	IF ( MsgRecBuffer[counter].MsgType = DATAREC AND   FIND(MsgRecBuffer[counter].Msg,  'NMEAS;MAC' ) = 4 ) AND ( FIND(MsgRecBuffer[counter].Msg,  'IDN' ) = 30) THEN
		StrSaveMacAdd:=MID(MsgRecBuffer[counter].Msg, 8 , 21);
		StrLoc:=33;
		Str := MID(MsgRecBuffer[counter].Msg, 1 , StrLoc);
		WHILE (SysStrCmp(Str,';')<>0 AND StrLoc<=255) DO (*Cerco il numero IDN e lo memorizzo in StrSaveID dopo il while*)
			StrLoc:=StrLoc+1;
			Str := MID(MsgRecBuffer[counter].Msg, 1 , StrLoc);
		END_WHILE
		StrSaveID:=MID(MsgRecBuffer[counter].Msg, StrLoc-33 , 33);
		index:=1;
		WHILE (index<=MAX_LUXNUM) AND (SysStrCmp(TabListLux[index].StMacAdd,  StrSaveMacAdd) <> 0)   DO (*diego setting *)
			index:= index +1;
		END_WHILE
		IF index<=MAX_LUXNUM AND STRING_TO_WORD(StrSaveID) >0 AND TabListLux[index].LuxID_Geolumen<>STRING_TO_WORD(StrSaveID)  THEN
			TabListLux[index].xCoupled := TRUE; (*Indico che ho accoppiato l'ID con il mac address*)
			TabListLux[index].LuxID_Geolumen:=STRING_TO_WORD(StrSaveID); (*Salvo l'ID accoppiato al mac address - info che sarà poi da spedire al server*)
			LuxElement[index].ID := TabListLux[index].LuxNumber; (*  copio id del lux nella tabella delle variabili dei lux *)
			IF LuxElement[index].CTRL_MODE = 2 THEN
				(* init astro *)
				ASTR[index](ID:= LuxElement[index].ID, localTime:=Sys.Time_CT_DT);
				ASTR_CONFIG[index].ID:=ASTR[index].ID;
			END_IF
			LuxGeolumenNodes[index].ID_Geolumen:=TabListLux[index].LuxID_Geolumen;
			LuxGeolumenNodes[index].ID_Lux:=TabListLux[index].LuxNumber;
			LuxGeolumenNodes[index].MAX_RETRY_NO_FEEDBACK:=MAX_RETRY_NO_FEEDBACK_GEOLUMEN_NODES;
			LuxGeolumenNodes[index].MAX_RETRY_STATUS_NOT_ALIGNED:=MAX_RETRY_STATUS_NOT_ALIGNED_GEOLUMEN_NODES;

			(*aggiorno stato*)
			parseNodeStatus(statusNodeMessage:=MsgRecBufferPtr^[counter].Msg);
			IF idNode>=1 AND idNode<=MAX_LUXNUM THEN
				tmpIndex:=getGeolumenNodeByGeolumenId (idNode);
				IF(tmpIndex>0 AND tmpIndex<=MAX_LUXNUM) THEN
					LuxGeolumenNodes[tmpIndex](feedbackState:=state); LuxGeolumenNodes[tmpIndex].updateFeedbackState();
				END_IF
			END_IF
		END_IF
	END_IF

	IF ( MsgRecBuffer[counter].MsgType = MED AND   FIND(MsgRecBuffer[counter].Msg,  'NMEASMED;MAC' ) = 4 ) AND ( FIND(MsgRecBuffer[counter].Msg,  'IDN' ) = 33) THEN
		StrSaveMacAdd:=MID(MsgRecBuffer[counter].Msg, 8 , 24);
		StrLoc:=36;
		Str := MID(MsgRecBuffer[counter].Msg, 1 , StrLoc);
		WHILE (SysStrCmp(Str,';')<>0 AND StrLoc<=255) DO (*Cerco il numero IDN e lo memorizzo in StrSaveID dopo il while*)
			StrLoc:=StrLoc+1;
			Str := MID(MsgRecBuffer[counter].Msg, 1 , StrLoc);
		END_WHILE
		StrSaveID:=MID(MsgRecBuffer[counter].Msg, StrLoc-36 , 36);
		index:=1;
		WHILE (index<=MAX_LUXNUM) AND (SysStrCmp(TabListLux[index].StMacAdd,  StrSaveMacAdd) <> 0)   DO (*diego setting *)
			index:= index +1;
		END_WHILE
		IF index<=MAX_LUXNUM AND STRING_TO_WORD(StrSaveID) >0 AND TabListLux[index].LuxID_Geolumen<>STRING_TO_WORD(StrSaveID)  THEN
			TabListLux[index].xCoupled := TRUE; (*Indico che ho accoppiato l'ID con il mac address*)
			TabListLux[index].LuxID_Geolumen:=STRING_TO_WORD(StrSaveID); (*Salvo l'ID accoppiato al mac address - info che sarà poi da spedire al server*)
			LuxElement[index].ID := TabListLux[index].LuxNumber; (*  copio id del lux nella tabella delle variabili dei lux *)
			IF LuxElement[index].CTRL_MODE = 2 THEN
				(* init astro *)
				ASTR[index](ID:= LuxElement[index].ID, localTime:=Sys.Time_CT_DT);
				ASTR_CONFIG[index].ID:=ASTR[index].ID;
			END_IF
			LuxGeolumenNodes[index].MAX_RETRY_NO_FEEDBACK:=MAX_RETRY_NO_FEEDBACK_GEOLUMEN_NODES;
			LuxGeolumenNodes[index].MAX_RETRY_STATUS_NOT_ALIGNED:=MAX_RETRY_STATUS_NOT_ALIGNED_GEOLUMEN_NODES;
			LuxGeolumenNodes[index].ID_Geolumen:=TabListLux[index].LuxID_Geolumen;
			LuxGeolumenNodes[index].ID_Lux:=TabListLux[index].LuxNumber;
		END_IF
	END_IF
END_ACTION
ACTION SendAuth:
(*...per compabilità indicizzazione Renato...*)
i:=ArrayPos-1;
IF(i<0) THEN i:=0; END_IF

(*TimerCmdAdd(IN:=NOT TimerCmdAdd.Q,PT:=T#5m);
IF TimerCmdAdd.Q THEN
	FOR x:= 1 TO MAX_LUXNUM DO
		TabListLuxSendAuth[x]:=0;
	END_FOR
END_IF*)


(*IF MsgRecBuffer[i].MsgType = REQAUTH0  THEN
	MacStr:=MID(MsgRecBuffer[i].Msg, 8, 23); (*Isolo la sottostringa del Mac address - es. 0046CD12*)

		FOR x:= 1 TO MAX_LUXNUM DO
			IF SysStrCmp(MacStr, TabListLux[x].StMacAdd) = 0 AND TabListLux[x].LuxID_Geolumen=0 AND TabListLuxSendAuth[x]<1 THEN
				TabListLuxSendAuth[x]:=TabListLuxSendAuth[x]+1;
				 (*spedisci autorizzazione   CMD_ADD_NODE:21:36096:70:50744$0D$0A  *)
				StrToSend:=CONCAT('LST_ADD_NODE:21,36096,', WORD_TO_STRING(TabListLux[x].MacAddH) );
				StrToSend:=CONCAT(StrToSend, ',');
				StrToSend:=CONCAT(StrToSend,  WORD_TO_STRING(TabListLux[x].MacAddL) );
				StrToSend:=CONCAT(StrToSend,  '$R' );
				(*SendData(pTxData:=ADR(StrToSend));*)
				SendDataQueue(pTxData:=ADR(StrToSend));
				SendDataQueue.addMessage();
				MsgRecBuffer[i].MsgType:=COMPLETED;
				x:=  MAX_LUXNUM+1;
			END_IF
		END_FOR

END_IF*)
END_ACTION
ACTION sendGlobalOff:
SendString := setGlobalOFF;
SendDataQueue(pTxData:=ADR(SendString));
SendDataQueue.addMessage();
END_ACTION
ACTION sendGlobalON:
SendString := setGlobalON;
SendDataQueue(pTxData:=ADR(SendString));
SendDataQueue.addMessage();
END_ACTION
ACTION updateNetworkTime:
(* creazione ed invio comando per settare orario della rete *)

StrMin:=BYTE_TO_STRING(Sys.Time_Min);
IF  Sys.Time_Min<=9 THEN
	StrMin := CONCAT('0',StrMin);
END_IF
StrMin:=MID(STR:=StrMin, LEN:=2, POS:= 1);
StrHour:=BYTE_TO_STRING(Sys.Time_Hour);
IF Sys.Time_Hour<=9 THEN
	StrHour := CONCAT('0',StrHour);
END_IF
StrHour:=MID(STR:=StrHour, LEN:=2, POS:= 1);

SendString := 'NWK_TIME_SET=$R';
SendString :=INSERT (SendString,StrHour,13);
SendString :=INSERT (SendString,':',15);
SendString :=INSERT (SendString,StrMin,16);

SendDataQueue(pTxData:=ADR(SendString));
SendDataQueue.addMessage();
END_ACTION

(* POU GeoLumenWrapping/SendDataQueue, ST *)
FUNCTION_BLOCK SendDataQueue
VAR CONSTANT
	QUEUE_SIZE:DWORD:=5000;
END_VAR
VAR_INPUT
	pTxData: POINTER TO STRING;
END_VAR
VAR_OUTPUT
	StrToSend: STRING;
	toBeSent : WORD:=0;
END_VAR
VAR
	writeIndex:DWORD:=0;
	readIndex:DWORD:=0;
	pRecStr 	: POINTER TO STRING(255);
	queue: ARRAY[1..QUEUE_SIZE] OF STRING(255);

END_VAR
;
END_FUNCTION_BLOCK
ACTION addMessage:
writeIndex:=((writeIndex+1) MOD (QUEUE_SIZE+1))+(writeIndex+1)/(QUEUE_SIZE+1);

queue[writeIndex]:=pTxData^;

IF(toBeSent<QUEUE_SIZE) THEN
	toBeSent:=toBeSent+1;
ELSE

	toBeSent:=1;

END_IF
END_ACTION
ACTION getMessage:
IF(toBeSent >0) THEN

	readIndex:=((readIndex+1) MOD (QUEUE_SIZE+1))+(readIndex+1)/(QUEUE_SIZE+1);

	StrToSend:=queue[readIndex];

	IF(toBeSent >0) THEN
		toBeSent:=toBeSent-1;
	END_IF

END_IF
END_ACTION
ACTION saveQueueToFile:
GeolumenSaveSendBuffer(ADR(QUEUE));
END_ACTION

(* POU GeoLumenWrapping/GeolumenSaveSendBuffer, ST *)
FUNCTION GeolumenSaveSendBuffer  : BOOL
VAR CONSTANT
	MY_QUEUE_SIZE:WORD:=5000;
END_VAR
VAR_INPUT
	queue:POINTER TO ARRAY[1..MY_QUEUE_SIZE] OF STRING(255);
END_VAR
VAR
	hName : STRING(255) :='SENDBUFF.TXT';
	hFile	 : DWORD;
	i	 : INT;
	line:STRING(255):='';
	tmp:STRING(8):='';
	macString:STRING(8);
	count:INT:=0;
	refCount:INT:=0;
END_VAR
hName:=CONCAT(FilesPath ,hName);
hFile:=SysFileOpen(hName,'w');
IF hFile<>0 THEN
	FOR i := 1 TO MY_QUEUE_SIZE  DO
		IF  SysStrCmp(queue^[i],'') <> 0  THEN
			line:=queue^[i];
			line:=CONCAT(line,'$N');
			SysFileWrite(hFile, ADR(line),LEN(line));
		END_IF
	END_FOR
	SysFileClose(hFile);
END_IF
END_FUNCTION

(* POU GeoLumenWrapping/getGeolumenNodeByGeolumenId, ST *)
FUNCTION getGeolumenNodeByGeolumenId : INT
VAR_INPUT
	GeolumenId : INT;
END_VAR

VAR
	I : INT;
END_VAR
getGeolumenNodeByGeolumenId:=-1;
FOR I:=1 TO MAX_LUXNUM DO
	IF (LuxGeolumenNodes[i].ID_Geolumen = GeolumenId) THEN getGeolumenNodeByGeolumenId :=i; RETURN; END_IF
END_FOR
END_FUNCTION

(* POU GeoLumenWrapping/isGeolumenNodesOffDuringDay, ST *)
FUNCTION_BLOCK isGeolumenNodesOffDuringDay
VAR_OUTPUT
	isGeolumenNodesOffDuringDay:BOOL;
END_VAR
VAR
	maxDT:DT;
	i:INT;
END_VAR
FOR i:=1 TO MAX_LUXNUM DO
	IF LuxElement[i].ID <> i THEN
		IF LuxGeolumenNodes[i].lastSeen > maxDT THEN
			maxDT:=LuxGeolumenNodes[i].lastSeen;
		END_IF
	END_IF
END_FOR

isGeolumenNodesOffDuringDay:=maxDT-Sys.Time_CT_DT > T#5m AND ( Sys.Time_CT_DT  > astroGen.timeEnd AND  Sys.Time_CT_DT  < astroGen.timeStart);
END_FUNCTION_BLOCK

(* POU GeoLumenWrapping/LuxGeolumenDiagnostics, ST *)
FUNCTION_BLOCK LuxGeolumenDiagnostics
VAR_INPUT
	turnOnRequest:BOOL;
	turnOffRequest:BOOL;
	restoreAllRequest:BOOL;
	executeCommandRequest:BOOL;
	executeCommandSetRequest:BOOL;
	executeCommandGetRequest:BOOL;
	executeCommandGetIDByMACRequest:BOOL;
	executeCommandGetMACByIDRequest:BOOL;
	executeCommandResetRequest:BOOL;
	executeCommandSaveToFileRequest:BOOL;
	executeCommandLoadFromFileRequest:BOOL;
	executeCommandSaveMsgBuffRequest:BOOL;
	executeCommandSaveSendBuffRequest:BOOL;
	executeCommandSaveNodeStatusRequest:BOOL;
	executeSendAuthAllRequest:BOOL;

	commandSetID:WORD;
	commandGetID:STRING(10):='';
	commandSetDIMM:INT;
	commandGetIDByMac:DWORD;
	commandGetIDByMacResult:DWORD;
	commandGetMacByID:WORD	;
	commandGetMacByIDResult:DWORD;
	diagnosticCommand:STRING(255):='';
	MacStr	: STRING (8);
	x:INT;
	StrToSend	:STRING(255);
END_VAR
VAR CONSTANT
	DELAY_FOR_LOG_EV:TIME:=T#200ms;
END_VAR
VAR
	LuxCount:WORD:=1;
	COUNT:INT:=0;
	I:INT:=0;
	TimerOnAll:TON;
	TimerOffAll:TON;
	TimerRestoreAll:TON;
END_VAR
IF restoreAllRequest THEN
	restoreAllStep();
END_IF
IF turnOnRequest THEN
	turnOnAllStep();
END_IF
IF turnOffRequest THEN
	turnOffAllStep();
END_IF
IF executeCommandRequest THEN
	executeCommand();
	executeCommandRequest:=FALSE;
END_IF
IF executeCommandSetRequest THEN
	executeSetCommand();
	executeCommandSetRequest:=FALSE;
END_IF
IF executeCommandGetRequest THEN
	executeGetCommand();
	executeCommandGetRequest:=FALSE;
END_IF
IF executeCommandGetIDByMACRequest THEN
	executeGetCommandIDByMAC();
	executeCommandGetIDByMACRequest:=FALSE;
END_IF
IF executeCommandGetMACByIDRequest THEN
	executeGetCommandMACByID();
	executeCommandGetMACByIDRequest:=FALSE;
END_IF
IF executeCommandResetRequest THEN
	executeCommandReset();
	executeCommandResetRequest :=FALSE;
END_IF
IF executeCommandSaveToFileRequest THEN
	GeolumenSaveTabListLux();
	executeCommandSaveToFileRequest  :=FALSE;
END_IF
IF executeCommandLoadFromFileRequest THEN
	GeolumenLoadTabListLux();
	executeCommandLoadFromFileRequest  :=FALSE;
END_IF
IF executeCommandSaveMsgBuffRequest THEN
	GeolumenSaveMsgBuff();
	executeCommandSaveMsgBuffRequest :=FALSE;
END_IF

IF executeCommandSaveSendBuffRequest THEN
	SendDataQueue.saveQueueToFile();
	executeCommandSaveSendBuffRequest :=FALSE;
END_IF


IF executeCommandSaveNodeStatusRequest THEN
	GeolumenSaveNodeStatus();
	executeCommandSaveNodeStatusRequest :=FALSE;
END_IF

IF executeSendAuthAllRequest THEN
	sendAuthAll();
	executeSendAuthAllRequest:=FALSE;
END_IF
END_FUNCTION_BLOCK
ACTION executeCommand:
IF FIND(diagnosticCommand,'$R') <1 THEN diagnosticCommand:=CONCAT(diagnosticCommand,'$R'); END_IF
SendDataQueue(pTxData:=ADR(diagnosticCommand));
SendDataQueue.addMessage();
END_ACTION
ACTION executeCommandReset:
diagnosticCommand:='CMD_SW_RESET$R';
SendDataQueue(pTxData:=ADR(diagnosticCommand));
SendDataQueue.addMessage();
diagnosticCommand:='CMD_AUTHORISE=0$R';
SendDataQueue(pTxData:=ADR(diagnosticCommand));
SendDataQueue.addMessage();
END_ACTION
ACTION executeGetCommand:
diagnosticCommand:='NDE_GET_STATUS=x$R';
diagnosticCommand:=REPLACE_ALL(diagnosticCommand,'x',commandGetID);

SendDataQueue(pTxData:=ADR(diagnosticCommand));
SendDataQueue.addMessage();
END_ACTION
ACTION executeGetCommandIDByMAC:
FOR LuxCount:=1 TO  MAX_LUXNUM DO
	IF  TabListLux[LuxCount].MacAdd<>0 AND TabListLux[LuxCount].MacAdd=commandGetIDByMac THEN
			commandGetIDByMacResult:=TabListLux[LuxCount].LuxNumber;
			RETURN;
	END_IF
END_FOR
END_ACTION
ACTION executeGetCommandMACByID:
FOR LuxCount:=1 TO  MAX_LUXNUM DO
	IF  TabListLux[LuxCount].LuxNumber<>0 AND TabListLux[LuxCount].LuxNumber=commandGetMacByID THEN
		commandGetMacByIDResult:=TabListLux[LuxCount].MacAdd;
		RETURN;
	END_IF
END_FOR
END_ACTION
ACTION executeSetCommand:
FOR i:=1 TO MAX_LUXNUM DO
		IF LuxElement[i].ID=commandSetID THEN

			IF(commandSetDIMM>0) THEN
					LuxElement [i] . CTRL_MODE := 1 ; (*// Set to manuale on con dimm*)
					LuxElement [i].DimmingValForManual:=commandSetDIMM;
			ELSE
					LuxElement [i] . CTRL_MODE := 0 ; (*// Set to manuale off*)
					LuxElement [i].DimmingValForManual:=0;
			END_IF

			LuxElement [  i  ] (     WORKINGTIME := GlobalWorkingTime [ i ] ,
			POWERONCYCLES:= GlobalPowerOnCycles [  i  ] ,
			ENERGYCOUNTER :=GlobalEnergyCounter [  i ] ,
			ENERGYCOUNTER_T :=GlobalEnergyCounter_t [  i  ] ,
									CtrlExton := KEYON ) ;
		END_IF
END_FOR
END_ACTION
ACTION restoreAllStep:
TimerRestoreAll(IN:=NOT TimerRestoreAll.Q,PT:=DELAY_FOR_LOG_EV);

	IF  TimerRestoreAll.Q THEN

		IF LuxElement[LuxCount].ID <> 0 THEN
			LuxElement [  LuxCount ] . CTRL_MODE := LuxElement [ LuxCount] . CTRL_MODE_backUp ;
			LuxElement [  LuxCount ] (     WORKINGTIME := GlobalWorkingTime [ LuxCount ] ,
							POWERONCYCLES :=
							GlobalPowerOnCycles [ LuxCount ] ,
							ENERGYCOUNTER := GlobalEnergyCounter [ LuxCount ] ,
							ENERGYCOUNTER_T :=
							GlobalEnergyCounter_t [ LuxCount ] ,
							CtrlExton := KEYON ) ;
		END_IF

		LuxCount:=LuxCount+1;
	END_IF


IF  LuxCount>MAX_LUXNUM  THEN
	LuxCount:=1;
	restoreAllRequest:=FALSE;
END_IF
END_ACTION
ACTION sendAuthAll:
	FOR x:= 1 TO MAX_LUXNUM DO
		IF TabListLuxSendAuth[x]<1 THEN

			TabListLuxSendAuth[x]:=TabListLuxSendAuth[x]+1;

			IF GEOLUMEN_COORD_VERSION = 1 THEN

				StrToSend:=CONCAT('CMD_ADD_NODE:21:36096:', WORD_TO_STRING(TabListLux[x].MacAddH) );
				StrToSend:=CONCAT(StrToSend, ':');
				StrToSend:=CONCAT(StrToSend,  WORD_TO_STRING(TabListLux[x].MacAddL) );
				StrToSend:=CONCAT(StrToSend,  '$R' );

			ELSIF GEOLUMEN_COORD_VERSION = 2 THEN

				StrToSend:=CONCAT('LST_ADD_NODE:21,36096,', WORD_TO_STRING(TabListLux[x].MacAddH) );
				StrToSend:=CONCAT(StrToSend, ',');
				StrToSend:=CONCAT(StrToSend,  WORD_TO_STRING(TabListLux[x].MacAddL) );
				StrToSend:=CONCAT(StrToSend,  '$R' );
			END_IF

			SendDataQueue(pTxData:=ADR(StrToSend));
			SendDataQueue.addMessage();

		END_IF

	END_FOR
END_ACTION
ACTION turnOffAllStep:
TimerOffAll(IN:=NOT TimerOffAll.Q,PT:=DELAY_FOR_LOG_EV);

	IF  TimerOffAll.Q THEN

			IF LuxElement[LuxCount].ID <> 0  THEN
					LuxElement [ LuxCount ] . CTRL_MODE := 0 ; (*// Set to manuale OFF *)
					LuxElement [ LuxCount ].DimmingValForManual:=0;
					LuxElement [ LuxCount ] (     WORKINGTIME := GlobalWorkingTime [ LuxCount ] ,
									POWERONCYCLES:= GlobalPowerOnCycles [ LuxCount ] ,
									ENERGYCOUNTER :=GlobalEnergyCounter [ LuxCount ] ,
									ENERGYCOUNTER_T :=GlobalEnergyCounter_t [ LuxCount ] ,
									CtrlExton := KEYON ) ;
			END_IF

				LuxCount:=LuxCount+1;
	END_IF



IF  LuxCount>MAX_LUXNUM  THEN
	LuxCount:=1;
	turnOffRequest:=FALSE;
END_IF
END_ACTION
ACTION turnOnAllStep:
TimerOnAll(IN:=NOT TimerOnAll.Q,PT:=DELAY_FOR_LOG_EV);

	IF  TimerOnAll.Q THEN

				IF LuxElement[LuxCount].ID <> 0 THEN
					LuxElement [ LuxCount  ] . CTRL_MODE := 1 ; (*// Set to manuale ON *)
					LuxElement [ LuxCount ].DimmingValForManual:=LuxElement [ LuxCount ].MAX_DIMM_VALUE;
					LuxElement [ LuxCount] (     WORKINGTIME := GlobalWorkingTime [ LuxCount ] ,
									POWERONCYCLES:= GlobalPowerOnCycles [ LuxCount ] ,
									ENERGYCOUNTER :=GlobalEnergyCounter [ LuxCount ] ,
									ENERGYCOUNTER_T :=GlobalEnergyCounter_t [ LuxCount ] ,
									CtrlExton := KEYON ) ;
				END_IF

				LuxCount:=LuxCount+1;

	END_IF

IF  LuxCount>MAX_LUXNUM  THEN
	LuxCount:=1;
	turnOnRequest:=FALSE;
END_IF
END_ACTION

(* POU GeoLumenWrapping/GeolumenSaveTabListLux, ST *)
FUNCTION GeolumenSaveTabListLux  : BOOL
VAR
	hName : STRING(255) :='TABLISTLUX.TXT';
	hFile	 : DWORD;
	i	 : INT;
	line:STRING(255):='';
	tmp:STRING(8):='';
	macString:STRING(8);

END_VAR
hName:=CONCAT(FilesPath ,hName);
hFile:=SysFileOpen(hName,'w');
IF hFile<>0 THEN
	FOR i := 1 TO MAX_LUXNUM  DO
			line:=CONCAT(DWORD_TO_STRING(TabListLux[i].LuxNumber),',');
			line:=CONCAT(line,DWORD_TO_STRING(TabListLux[i].LuxID_Geolumen));
			line:=CONCAT(line,',');
			tmp:=DWORD_TO_STRH(TabListLux[i].MacAdd);
			line:=CONCAT(line,tmp);
			line:=CONCAT(line,';');
			IF i<MAX_LUXNUM THEN line:=CONCAT(line,'$R$N'); END_IF
			SysFileWrite(hFile, ADR(line),LEN(line));
	END_FOR
	SysFileClose(hFile);
END_IF
END_FUNCTION

(* POU GeoLumenWrapping/GeolumenLoadTabListLux, ST *)
FUNCTION GeolumenLoadTabListLux  : BOOL
VAR
	hName : STRING(255) :='TABLISTLUX.TXT';
	hFile	 : DWORD;
	i	 : INT;
	line:STRING(255):='';
	tmp:STRING(8):='';
	macString:STRING(8);
	stringLuxNumber:STRING(255);
	stringSep:STRING(255);
END_VAR
(*hName:=CONCAT(FilesPath ,hName);
hFile:=SysFileOpen(hName,'r');
IF hFile<>0 THEN
	FOR i := 1 TO MAX_LUXNUM  DO
			SysFileRead(hFile,ADR(stringLuxNumber), SIZEOF(TabListLux[i].LuxNumber));
			line:=CONCAT(DWORD_TO_STRING(TabListLux[i].LuxNumber),',');
			line:=CONCAT(line,DWORD_TO_STRING(TabListLux[i].LuxID_Geolumen));
			line:=CONCAT(line,',');
			tmp:=DWORD_TO_STRH(TabListLux[i].MacAdd);
			line:=CONCAT(line,tmp);
			line:=CONCAT(line,';');
			IF i<MAX_LUXNUM THEN line:=CONCAT(line,'$R$N'); END_IF
			SysFileWrite(hFile, ADR(line),LEN(line));
	END_FOR
	SysFileClose(hFile);
END_IF*)
;
END_FUNCTION

(* POU GeoLumenWrapping/GeolumenSaveMsgBuff, ST *)
FUNCTION GeolumenSaveMsgBuff  : BOOL
VAR
	hName : STRING(255) :='MSGBUFF.TXT';
	hFile	 : DWORD;
	i	 : INT;
	line:STRING(255):='';
	tmp:STRING(8):='';
	macString:STRING(8);
	count:INT:=0;
	refCount:INT:=0;
END_VAR
hName:=CONCAT(FilesPath ,hName);
hFile:=SysFileOpen(hName,'w');
IF hFile<>0 THEN
	FOR i := 0 TO MAX_ARRAY_MSG DO
			line:='';
			line:=CONCAT(MsgRecBuffer[i].Msg,'$R$N');
			SysFileWrite(hFile, ADR(line),LEN(line));
	END_FOR
	SysFileClose(hFile);
END_IF
END_FUNCTION

(* POU GeoLumenWrapping/GeolumenSaveNodeStatus, ST *)
FUNCTION GeolumenSaveNodeStatus  : BOOL
VAR
	hName : STRING(255) ;
	hFile	 : DWORD;
	i	 : INT;
	line:STRING(255):='';
	tmp:STRING(8):='';
	macString:STRING(8);

END_VAR
hName:=CONCAT(FilesPath ,'snapshot/');
hName:=CONCAT(hName ,DWORD_TO_STRING(Plant_SN));
hName:=CONCAT(hName ,'_');
hName:=CONCAT(hName ,'nodeStatus_');
hName:=CONCAT(hName ,WORD_TO_STRING(SYS.Time_Year));
hName:=CONCAT(hName ,SEL(SYS.Time_Month>=10, CONCAT('0',WORD_TO_STRING(SYS.Time_Month)) , WORD_TO_STRING(SYS.Time_Month)));
hName:=CONCAT(hName ,SEL(SYS.Time_Day>=10, CONCAT('0',WORD_TO_STRING(SYS.Time_Day)) , WORD_TO_STRING(SYS.Time_Day)));
hName:=CONCAT(hName ,'_');
hName:=CONCAT(hName ,SEL(SYS.Time_Hour>=10, CONCAT('0',WORD_TO_STRING(SYS.Time_Hour)) , WORD_TO_STRING(SYS.Time_Hour)));
hName:=CONCAT(hName ,SEL(SYS.Time_Min>=10, CONCAT('0',WORD_TO_STRING(SYS.Time_Min)) , WORD_TO_STRING(SYS.Time_Min)));
hName:=CONCAT(hName ,'.txt');
hFile:=SysFileOpen(hName,'w');
IF hFile<>0 THEN
	FOR i := 1 TO MAX_LUXNUM  DO
			line:=CONCAT(DWORD_TO_STRING(TabListLux[i].LuxNumber),',');
			line:=CONCAT(line,DWORD_TO_STRING(TabListLux[i].LuxID_Geolumen));
			line:=CONCAT(line,',');
			tmp:=DWORD_TO_STRH(TabListLux[i].MacAdd);
			line:=CONCAT(line,tmp);
			SysFileWrite(hFile, ADR(line),LEN(line));

			line:=CONCAT(',',WORD_TO_STRING(LuxGeolumenNodes[i].feedbackState.LqiLast));
			line:=CONCAT(line,',');
			line:=CONCAT(line,WORD_TO_STRING(LuxGeolumenNodes[i].feedbackState.LqiAvg));
			line:=CONCAT(line,',');
			line:=CONCAT(line,WORD_TO_STRING(LuxGeolumenNodes[i].feedbackState.LqiMin));
			line:=CONCAT(line,',');
			line:=CONCAT(line,WORD_TO_STRING(LuxGeolumenNodes[i].feedbackState.LqiMax));
			SysFileWrite(hFile, ADR(line),LEN(line));

			line:=CONCAT(',',DT_TO_STRING(LuxGeolumenNodes[i].lastSeen));
			line:=CONCAT(line,',');
			line:=CONCAT(line, DWORD_TO_STRING(LuxGeolumenNodes[i].retryStatusNotAligned));
			line:=CONCAT(line,',');
			line:=CONCAT(line, DT_TO_STRING(LuxGeolumenNodes[i].echoLastSeen));
			line:=CONCAT(line,',');
			line:=CONCAT(line, WORD_TO_STRING(LuxElement[I].Lux_StateAnalog));
			line:=CONCAT(line,',');
			line:=CONCAT(line, WORD_TO_STRING(LuxGeolumenChangeFlag[i]));
			line:=CONCAT(line,',');
			line:=CONCAT(line, BOOL_TO_STRING(LuxGeolumenNodesAlignFlags[i]));
			SysFileWrite(hFile, ADR(line),LEN(line));


			line:=CONCAT(',',SEL(LEN(LuxGeolumenNodes[i].lastPar)>0, 'N/A', LuxGeolumenNodes[i].lastPar));
			SysFileWrite(hFile, ADR(line),LEN(line));

			line:=';';
			IF i<MAX_LUXNUM THEN line:=CONCAT(line,'$R$N'); END_IF
			SysFileWrite(hFile, ADR(line),LEN(line));
	END_FOR
	SysFileClose(hFile);
END_IF
END_FUNCTION

(* POU GeoLumenWrapping/isCoordinatorBooted, ST *)
FUNCTION isCoordinatorBooted : BOOL
VAR
END_VAR
(*isCoordinatorBooted:=(SYS.Time_CT_DT- PLC_START_TIME)>T#10m;*)
isCoordinatorBooted:=TRUE;
END_FUNCTION

(* POU GeoLumenWrapping/isGeolumenEqualStatus, ST *)
FUNCTION isGeolumenEqualStatus : BOOL
VAR_INPUT
	desideredState: type_LuxGeolumenStatus;
	feedbackState: type_LuxGeolumenStatus;
END_VAR
VAR
END_VAR
isGeolumenEqualStatus:=(desideredState.ID_Geolumen=feedbackState.ID_Geolumen) AND
					  (desideredState.DimmValue_0=feedbackState.DimmValue_0) AND
 					  (desideredState.DimmValue_1=feedbackState.DimmValue_1) AND
					  (desideredState.DimmValue_2=feedbackState.DimmValue_2) ;
(*IF (desideredState.DimmValue_0 >0 OR desideredState.DimmValue_1 >0 OR desideredState.DimmValue_2 > 0) AND NOT (feedbackState.LampCurrent>0) THEN
	isGeolumenIEqualStatus:=FALSE;
END_IF
IF (desideredState.DimmValue_0 =0 AND desideredState.DimmValue_1 =0 AND desideredState.DimmValue_2 =0 ) AND feedbackState.LampCurrent>0 THEN
	isGeolumenIEqualStatus:=FALSE;
END_IF*)
END_FUNCTION

(* POU ClevergyUtils/TCP_Logger/LogTrig, ST *)
FUNCTION LogTrig : BOOL
VAR
	s1 : STRING(160);
	i  : BYTE;
END_VAR
(*---------------------------------------------------------------*)
	Logger_Head();
(*---------------------------------------------------------------*)

Plant_LogTrig();

(*---------------------------------------------------------------*)
	Logger_Send();
(*---------------------------------------------------------------*)
END_FUNCTION

(* POU ClevergyUtils/TCP_Logger/Logger_Head, ST *)
FUNCTION Logger_Head : BOOL
VAR
	s1 : STRING(160);
	i  : BYTE;
END_VAR
(* Create the header to transmit the logfile on the VPN according to internal protocol	*)
Logger.TLen:=0;

(* Set GET header *)
ADDSTRING(ADR(Logger.TData), ADR(Logger_GETSTART), Logger.TLen);

(* Insert Header *)
s1:=INSERT('ID=&V=1&D=',DWORD_TO_STRING(Plant_SN),3);		(* Insert plant ID after 3 characters, therefore after string
																'ID='	*)
s1:=CONCAT(s1,Sys.Time_LogString);							(* Add Data and Time	*)
s1:=CONCAT(s1,'&S=');

(* Check what to signal according to the flag: Alarm, Warning or everything OK	*)
IF Sys.Alarm THEN i:=2; ELSIF Sys.Warning THEN i:=1; ELSE i:=0; END_IF
s1:=CONCAT(s1,BYTE_TO_STRING(i));

ADDSTRING(ADR(Logger.TData), ADR(s1), Logger.TLen);
END_FUNCTION

(* POU ClevergyUtils/ADDSTRING, ST *)
FUNCTION ADDSTRING : BOOL (* Append string to a byte buffer *)
VAR_INPUT
	pTxData: POINTER TO BYTE;
	pString: POINTER TO BYTE;
END_VAR
VAR_IN_OUT
	TxLen: DINT;
END_VAR
VAR
END_VAR
(* Add a string starting from an offset ("TxLen") using pointer. Stop the add when the string to copy has a 0 as argument	*)
pTxData:=pTxData+TxLen;
WHILE pString^<>0 DO
	pTxData^:=pString^;
	pString:=pString+1;
	pTxData:=pTxData+1;
	TxLen:=TxLen+1;
END_WHILE
END_FUNCTION

(* POU PLANTCONFIG/Plant_LogTrig, ST *)
FUNCTION Plant_LogTrig : BOOL
VAR_INPUT
END_VAR
VAR
	i:INT;
END_VAR
(*richiedo di loggare da ora*)
SyncLogRequest:=TRUE;
timingLuxBase:=t#0m;
timingAstroBase:=t#1m30s;
logRowLux:=0;
logRowAstro:=0;

FOR i:=1 TO MAX_LOG_ROW DO

	TimerLogAstroSyncDone[I]:=FALSE;
	TimerLogLuxSyncDone[I]:=FALSE;

END_FOR
END_FUNCTION

(* POU ClevergyUtils/TCP_Logger/Logger_Send, ST *)
FUNCTION Logger_Send : BOOL
VAR
	hFile: 	DWORD;
	pos:	DWORD;
END_VAR
(* Finalize string *)
ADDSTRING(ADR(Logger.TData), ADR(Logger_GETEND), Logger.TLen);		(* Code that identifies the end of the "GET" log  *)

(* Read log position *)
pos:=SysFileGetSize(Logger_DataFile);								(* Get size in byte of the file	*)

(* Check log size, bckup and erase if no pending messages *)
IF pos>5000000(*5M*) THEN
	hFile:=SysFileOpen(Logger_IndexFile,'r');

	IF hFile=0 THEN							(* If "Logger_IndexFile" doesn't exist -> No pending messagge to be transmitted	*)
		SysFileDelete(Logger_DataFileOld);							(* Delete old log file (backup)	*)
		SysFileRename(Logger_DataFile,Logger_DataFileOld);			(* Rename new log file as "DataFileOld" (backup) *)
		pos:=0;
	ELSE
		SysFileClose(hFile);
	END_IF
END_IF
(* ^^^ Delete old backup file and if actual logger file is too big and all messagges have been transmitted, set it as backup *)

(* Write message on log file *)
hFile:=SysFileOpen(Logger_DataFile,'a');							(* Open in write mode, but new data ar added at the end *)

(* If no error occurs when opening the log file, write new data ("Logger.TData")	*)
IF hFile<>0 THEN
	SysFileWrite(hFile, ADR(Logger.TData), Logger.TLen);
	SysFileClose(hFile);
	warningHFileLogSend:=FALSE;
ELSE
	(*Sys.Warning:=TRUE;*)		(* Set a system warning	*)
	warningHFileLogSend:=TRUE;
END_IF


(* Check logger status *)
IF Logger.SendReq=FALSE THEN
	(* Set log position for recovery *)
	Logger.SendIdx:=pos;
	(* Copy message data *)
	MEMCPY(ADR(Logger.TData),ADR(Logger.SendData),DINT_TO_WORD(Logger.TLen));
	Logger.SendLen:=Logger.TLen;
	(* Trigger request *)
	Logger.SendReq:=TRUE;
ELSE
	(* Connection still busy, so it's not possible to send now data. Write the LoggerIndex file	*)
	(* Add message position+size in recovery indexes *)
	hFile:=SysFileOpen(Logger_IndexFile,'a');
	SysFileWrite(hFile, ADR(pos), SIZEOF(pos));
	SysFileWrite(hFile, ADR(Logger.TLen), SIZEOF(Logger.TLen));
	SysFileClose(hFile);
END_IF
END_FUNCTION

(* POU ClevergyUtils/MEMCPY, ST *)
FUNCTION MEMCPY:BOOL
VAR_INPUT
	pSourceAddress:POINTER TO ARRAY[1..2] OF BYTE;
	pDestinationAddress:POINTER TO ARRAY[1..2] OF BYTE;
	BytesToCopy:WORD;
END_VAR
VAR
END_VAR
WHILE (BytesToCopy > 0) DO
	pDestinationAddress^[1]:=pSourceAddress^[1]; (* copy bytes from source to destination *)
	pDestinationAddress:=ADR(pDestinationAddress^[2]); (* increment destination *)
	pSourceAddress:=ADR(pSourceAddress^[2]);(* increment source *)
	BytesToCopy:=BytesToCopy -1; (* decrement number of bytes to copy *)
END_WHILE
END_FUNCTION

(* POU ClevergyUtils/RTC_Update, ST *)
PROGRAM RTC_Update
VAR
	T: DT;
	TS: STRING;
	TS2: STRING;
	Hour: BYTE;
	Minute: BYTE;
END_VAR
(* Get RTC time *)
T:=SysRtcGetTime(TRUE);
Sys.Time_CT_DT:=T;

(* Calculate variables *)
TS:=DT_TO_STRING(T);								(* Convert a format DATA_AND_TIME into a string, with the following
														result: 'DT#YYYY-MM-DD-HH:MM'	*)

Sys.Time_LogString:=DELETE(STR:=TS, LEN:=3, POS:=1);	(* Delete 3 characters starting from character number 1, the first
															so it deletes 'DT#'	*)

(* Proceed as before to isolate Year, Month and Day and convert them into a number format	*)
TS2:=MID(STR:=TS, LEN:=4, POS:= 4); Sys.Time_Year 	:=STRING_TO_WORD(TS2);
Sys.Time_Year 	:=STRING_TO_WORD(TS2);
TS2:=MID(STR:=TS, LEN:=2, POS:= 9); Sys.Time_Month	:=STRING_TO_BYTE(TS2);
Sys.Time_Month	:=STRING_TO_BYTE(TS2);
TS2:=MID(STR:=TS, LEN:=2, POS:=12); Sys.Time_Day  	:=STRING_TO_BYTE(TS2);
Sys.Time_Day  	:=STRING_TO_BYTE(TS2);

Sys.Time_CT_Day:=(32*(Sys.Time_Month-1)+Sys.Time_Day-1);

(* Proceed as before to isolate Hour and minute and convert them into a number format	*)
TS2:=MID(STR:=TS, LEN:=2, POS:=15); HOUR			:=STRING_TO_BYTE(TS2);
HOUR :=STRING_TO_BYTE(TS2);
Sys.Time_Hour := STRING_TO_BYTE(TS2);
TS2:=MID(STR:=TS, LEN:=2, POS:=18); MINUTE		 	:=STRING_TO_BYTE(TS2);
MINUTE :=STRING_TO_BYTE(TS2);
Sys.Time_Min:=STRING_TO_BYTE(TS2);

(* Calculate quarters of hour	*)
Sys.Time_CT_Quarter:=Hour*4+(Minute/15);
END_PROGRAM

(* POU PLANT_PROCESS/SCA_Proc, ST *)
PROGRAM SCA_Proc
VAR

	fCoord		:FLT_TAP;  (* geolumen coord STATUS *)
	(*SCA01_1	:	FLT_TAP;
	SCA01_2	:	FLT_TAP;
	SCA01_3	:	FLT_TAP;

	upd		:	BOOL;*)
END_VAR
(*### geolumen COORD Status Check ###*)
fCoord(IN:=COORD_STATUS);
IF fCoord.EVH THEN
	LogEv(EL_Log,EO_DOOR,1,1,'LIGHT_BOX_CLOSED');
END_IF
IF fCoord.EVL THEN
	LogEv(EL_Wrn,EO_DOOR,1,2,'LIGHT_BOX_OPENED');
END_IF

(***** SCA01 *****)
(*SCA01_1(IN:=SCA01_1_DI);
IF SCA01_1.EVL THEN LogEv(EL_Wrn,EO_SCA,1,1,'1'); upd:=TRUE; END_IF
IF SCA01_1.EVH THEN	LogEv(EL_Log,EO_SCA,1,2,'1'); upd:=TRUE; END_IF

SCA01_2(IN:=SCA01_2_DI);
IF SCA01_2.EVL THEN	LogEv(EL_Wrn,EO_SCA,1,1,'2'); upd:=TRUE; END_IF
IF SCA01_2.EVH THEN	LogEv(EL_Log,EO_SCA,1,2,'2'); upd:=TRUE; END_IF

SCA01_3(IN:=SCA01_3_DI);
IF SCA01_3.EVL THEN	LogEv(EL_Wrn,EO_SCA,1,1,'3'); upd:=TRUE; END_IF
IF SCA01_3.EVH THEN	LogEv(EL_Log,EO_SCA,1,2,'3'); upd:=TRUE; END_IF

IF upd THEN
	upd:=FALSE;
	Logger_Head();
	AddLogData();
	Logger_Send();
END_IF*)
;
END_PROGRAM
ACTION AddLogData:
(*Logger.s1:='&SCA01=';
Logger.s1:=CONCAT(Logger.s1,BYTE_TO_STRING(BOOL_TO_BYTE(SCA01_1.OUT))		); Logger.s1:=CONCAT(Logger.s1,';');
Logger.s1:=CONCAT(Logger.s1,BYTE_TO_STRING(BOOL_TO_BYTE(SCA01_2.OUT))		); Logger.s1:=CONCAT(Logger.s1,';');
Logger.s1:=CONCAT(Logger.s1,BYTE_TO_STRING(BOOL_TO_BYTE(SCA01_3.OUT))		);
ADDSTRING(ADR(Logger.TData), ADR(Logger.s1), Logger.TLen);*)
;
END_ACTION

(* POU ClevergyUtils/FLT_TAP, ST *)
FUNCTION_BLOCK FLT_TAP
VAR_INPUT
	IN		: BOOL;
	TAP		: BYTE:=4;
	INITEV	: BOOL:=TRUE;
END_VAR
VAR_OUTPUT
	OUT		: BOOL;
	EVH		: BOOL;
	EVL		: BOOL;
END_VAR
VAR
	init	: BOOL:=FALSE;
	cnt		: BYTE;
END_VAR
EVH:=FALSE;
EVL:=FALSE;

(* This first IF is done only the first time the FB is called, to read the actual (startup) value of the element;
   After first iteration, "init" becomes true and this IF is always skipped, unless a reset occurs	*)
IF NOT init THEN
	init := TRUE;
	IF INITEV THEN
		OUT  := NOT IN;
		cnt  := TAP;
	ELSE
		OUT  := IN;
	END_IF
END_IF

(* Need "TAP" equals level before update "OUT"	*)
IF OUT<>IN THEN
	cnt:=cnt+1;
	IF cnt>TAP THEN
		OUT:=IN;
		cnt:=0;
		IF OUT THEN EVH:=TRUE; ELSE EVL:=TRUE; END_IF
	END_IF
ELSE
	cnt:=0;
END_IF
END_FUNCTION_BLOCK

(* POU ClevergyUtils/TCP_Logger/LogEv, ST *)
FUNCTION LogEv : BOOL
VAR_INPUT
	Level	: en_Logger_ErrLev;
	Object  : en_SYS_Objects;
	Index	: DWORD;
	Error	: WORD;
	Message : STRING;
END_VAR
VAR
	s1 : STRING(160);
	i  : INT;
END_VAR
(* Generates the log for the error revealed	*)

(* Execute error level operations *)
(*CASE Level OF
	EL_Wrn: 		Sys.Warning:=TRUE;
	EL_Alarm: 		Sys.Alarm  :=TRUE;
	EL_AlarmStop: 	Sys.Alarm  :=TRUE; (* GO TO STOP STATE!! *)
END_CASE*)

(*** Runtime memory for last 5 logs (it's a sort of backup)	***)
(* Fill lastlog list *)
s1:=CONCAT(Sys.Time_LogString,';Lev=');			(* Insert current data and time read at the beginning *)
s1:=CONCAT(s1,INT_TO_STRING(Level));			(* Insert error level	*)
s1:=CONCAT(s1,';Obj=');
s1:=CONCAT(s1,INT_TO_STRING(Object));			(* Insert object who generates the error	*)
s1:=CONCAT(s1,';Idx=');
s1:=CONCAT(s1,DWORD_TO_STRING(Index));			(* Insert ID of the object in the system	*)
s1:=CONCAT(s1,';Err=');
s1:=CONCAT(s1,WORD_TO_STRING(Error));			(* Insert specific error	*)

(* This is used to keep last 5 logs in memory	*)
Sys.LastLogs_Dat[Sys.LastLogs_Idx]:=s1;
Sys.LastLogs_Msg[Sys.LastLogs_Idx]:=Message;
Sys.LastLogs_Idx:=Sys.LastLogs_Idx+1;

IF Sys.LastLogs_Idx>5 THEN Sys.LastLogs_Idx:=0; END_IF	(* If log index reach the end of the array, restart the index (Set it to 0)	*)

(*---------------------------------------------------------------*)
	Logger_Head();
(*---------------------------------------------------------------*)

(* Insert ERR *)		(* Repeat previous steps to create the log has to be transmitted on the network	*)
IF Level = EL_Evt THEN
	s1:=CONCAT('&ERR=',INT_TO_STRING(Level-EL_Evt));
ELSE
	s1:=CONCAT('&ERR=',INT_TO_STRING(Level));
END_IF
s1:=CONCAT(s1,';');
s1:=CONCAT(s1,INT_TO_STRING(Object));
s1:=CONCAT(s1,';');
s1:=CONCAT(s1,DWORD_TO_STRING(Index));
s1:=CONCAT(s1,';');
s1:=CONCAT(s1,WORD_TO_STRING(Error));
s1:=CONCAT(s1,';');

ADDSTRING(ADR(Logger.TData), ADR(s1), Logger.TLen);		(* Add this part of the log to the previous one (the header)	*)
s1:=Message;
STR_NOSPACES(ADR(s1));									(* Check there are no blank spaces in the "Message"	*)
ADDSTRING(ADR(Logger.TData), ADR(s1), Logger.TLen);		(* Add error message to the rest of the log file	*)

(*---------------------------------------------------------------*)
	Logger_Send();
(*---------------------------------------------------------------*)
END_FUNCTION

(* POU ClevergyUtils/STR_NOSPACES, ST *)
FUNCTION STR_NOSPACES : BOOL (* Replace spaces and bad chars with allowed ones, used as HTTP-GET validator *)
VAR_INPUT
	pString: POINTER TO BYTE;
END_VAR
VAR
END_VAR
WHILE pString^<>0 DO
	IF pString^=16#20 (* space *) THEN pString^:=16#5F; (*'_'*) END_IF
	pString:=pString+1;
END_WHILE
END_FUNCTION

(* POU PLANT_PROCESS/SYS_Proc, ST *)
PROGRAM SYS_Proc
VAR
	fVPN_ST2		:FLT_TAP;  (* VPN STATUS *)
(*	fKEY_CT_ST		:FLT_TAP; (* DOOR01 - Porta primaria *)*)
(*	fKEY_SCT_ST		:FLT_TAP; (* DOOR02 - Porta secondaria *)*)

END_VAR
(*### VPN Status Check ###*)
fVPN_ST2(IN:=VPN_STATUS);
IF fVPN_ST2.EVH THEN
	LogEv(EL_Log,EO_VPN,1,3,'STATUS_UP');
END_IF
IF fVPN_ST2.EVL THEN
	LogEv(EL_Wrn,EO_VPN,1,4,'STATUS_DOWN');
END_IF
END_PROGRAM

(* POU ClevergyUtils/Utils/USRLED_Update, ST *)
PROGRAM USRLED_Update
VAR
	Status	:	BYTE;
END_VAR
Status := PlantStatus;
PlantStatus := 0;	(* Reset value *)

(* Plant status (Alarm, warning or everything ok) *)
IF Status = 2 THEN
	LED_SET_STATIC(diLed_No:=7, eColor:=2);
	RETURN;
ELSIF Status = 1 THEN
	LED_SET_BLINK(diLed_No:=7, timTime1:=T#500ms, timTime2:=T#500ms, eColor1:=0, eColor2:=3);
	RETURN;
END_IF

(* VPN status led signalling *)
IF VPN_ST2 = 0 THEN
	LED_SET_BLINK(diLed_No:=7, timTime1:=T#500ms, timTime2:=T#500ms, eColor1:=0, eColor2:=2);
	RETURN;
END_IF

(* ModBus status led signalling *)
IF MODB01.MB_MASTER.bInterfaceError <> 0 THEN
	LED_SET_BLINK(diLed_No:=7, timTime1:=T#1s, timTime2:=T#1s, eColor1:=0, eColor2:=2);
	RETURN;
END_IF

(* Main Siwtch or Interface *)
IF INT01 = 0 OR INT02 = 0 THEN
	LED_SET_BLINK(diLed_No:=7, timTime1:=T#2s, timTime2:=T#2s, eColor1:=0, eColor2:=2);
	RETURN;
END_IF

(* System status led signalling *)
CASE SYS.Status OF

	S_STARTUP:
				(* Orange static *)
				LED_SET_STATIC(diLED_No:=7, eColor:=3);

	S_RUNNING:
				(* Green static *)
				LED_SET_STATIC(diLED_No:=7, eColor:=1);

END_CASE
END_PROGRAM

(* POU ClevergyUtils/Utils Functions/AVERAGE_DINT, ST *)
FUNCTION_BLOCK AVERAGE_DINT
VAR_INPUT
	IN: 	DINT;
END_VAR
VAR_OUTPUT
	HI:		DINT;
	AVG:	DINT;
	LOW:	DINT;
	ERR:	BOOL;
END_VAR
VAR
	sum:	REAL;
	cnt:	WORD;
END_VAR
IF cnt>=65000 THEN
	ERR:=TRUE;
	Read();
	sum := sum - DINT_TO_REAL(AVG);
	cnt := cnt - 1;
END_IF

sum := sum + DINT_TO_REAL(IN);
cnt := cnt + 1;

IF IN<LOW THEN LOW:=IN; END_IF
IF IN>HI  THEN HI :=IN; END_IF
END_FUNCTION_BLOCK
ACTION Read:
AVG := REAL_TO_DINT(sum/cnt);
END_ACTION
ACTION Reset:
HI:=IN;
AVG:=IN;
LOW:=IN;
ERR:=FALSE;

sum:=DINT_TO_REAL(IN);
cnt:=1;
END_ACTION

(* POU ClevergyUtils/Utils Functions/AVERAGE_INT, ST *)
FUNCTION_BLOCK AVERAGE_INT
VAR_INPUT
	IN: 	INT;
END_VAR
VAR_OUTPUT
	HI:		INT;
	AVG:	INT;
	LOW:	INT;
	ERR:	BOOL;
END_VAR
VAR
	sum:	DINT;
	cnt:	WORD;
END_VAR
IF cnt>=65000 THEN
	ERR:=TRUE;
	Read();
	sum := sum - AVG;
	cnt := cnt - 1;
END_IF

sum := sum + IN;
cnt := cnt + 1;

IF IN<LOW THEN LOW:=IN; END_IF
IF IN>HI  THEN HI :=IN; END_IF
END_FUNCTION_BLOCK
ACTION Read:
AVG := DINT_TO_INT(sum/cnt);
END_ACTION
ACTION Reset:
HI:=IN;
AVG:=IN;
LOW:=IN;
ERR:=FALSE;

sum:=IN;
cnt:=1;
END_ACTION

(* POU ClevergyUtils/AVERAGE_T, ST *)
FUNCTION_BLOCK AVERAGE_T
VAR_INPUT
	IN: 	INT;
END_VAR
VAR_OUTPUT
	HI:		INT;
	AVG:	INT;
	LOW:	INT;
	ERR:	BOOL;
END_VAR
VAR
	sum:	DINT;
	cnt:	WORD;
END_VAR
IF cnt>=65000 THEN
	ERR:=TRUE;
	Read();
	sum := sum - AVG;
	cnt := cnt + 1;
END_IF

sum := sum + IN;
cnt := cnt + 1;

IF IN<LOW THEN  LOW:=IN; END_IF
IF IN>HI  THEN HI :=IN; END_IF
END_FUNCTION_BLOCK
ACTION Read:
AVG := DINT_TO_INT(sum/cnt);
END_ACTION
ACTION Reset:
HI:=IN;
AVG:=IN;
LOW:=IN;
ERR:=FALSE;

sum:=IN;
cnt:=1;
END_ACTION

(* POU ClevergyUtils/BUILD_16TO32_COPY, ST *)
FUNCTION BUILD_16TO32_COPY : DWORD
VAR_INPUT
		LSW	:	WORD;
		MSW	:	WORD;
END_VAR
VAR
		Op1	:	DWORD;
		Op2	:	DWORD;
END_VAR
Op1  := WORD_TO_DWORD(LSW);

Op2 := WORD_TO_DWORD(MSW);
Op2 := SHL(Op2, 16);

BUILD_16TO32_COPY := Op1 + Op2;
END_FUNCTION

(* POU ClevergyUtils/Utils Functions/CheckPlant, ST *)
FUNCTION CheckPlant : BOOL
VAR_INPUT
		Obj_Status_Log	:	BYTE;
END_VAR
VAR
END_VAR
IF Obj_Status_Log = 0 THEN RETURN; END_IF

IF PlantStatus = 2 THEN RETURN; END_IF

IF PlantStatus = 1 THEN
	IF Obj_Status_Log = 2 THEN
		PlantStatus := 2;
		RETURN;
	END_IF
END_IF

IF PlantStatus = 0 THEN
	PlantStatus := Obj_Status_Log;
	RETURN;
END_IF
END_FUNCTION

(* POU ClevergyUtils/clv_TONOF, ST *)
FUNCTION_BLOCK clv_TONOF
VAR_INPUT
	IN		: BOOL;
	PT_ON	: TIME; (* time to pass, before OUT is set *)
	PT_OF	: TIME; (* time to pass, before OUT is reset *)
END_VAR
VAR_OUTPUT
	OUT		: BOOL;
END_VAR
VAR
	timer	: TON;
END_VAR
IF IN<>OUT THEN
	timer(IN:=TRUE,PT:=SEL(IN,PT_OF,PT_ON));
	IF timer.Q THEN OUT:=IN; END_IF
ELSE
	timer(IN:=FALSE);
END_IF
END_FUNCTION_BLOCK

(* POU ClevergyUtils/COPY_32SWAP16, ST *)
FUNCTION COPY_32SWAP16:BOOL
VAR_INPUT
	pSourceAddress		:POINTER TO ARRAY[1..2] OF WORD;
	pDestinationAddress	:POINTER TO ARRAY[1..2] OF WORD;
END_VAR
VAR
END_VAR
pDestinationAddress^[1]:=pSourceAddress^[2];
pDestinationAddress^[2]:=pSourceAddress^[1];
END_FUNCTION

(* POU ClevergyUtils/Utils/CSV_Log, ST *)
FUNCTION CSV_Log : BOOL
VAR_INPUT
END_VAR
VAR CONSTANT
	LogFileName:STRING:='S:\LOGS_ID4V3.CSV';
END_VAR
VAR
	s1 : STRING(256);
	hFile: 	DWORD;
END_VAR
(* Check file presence *)
hFile:=SysFileOpen(LogFileName,'r');
IF hFile=0 THEN
	(*** File not exist *** Create file and write header *)
	hFile:=SysFileOpen(LogFileName,'w');
	IF hFile<>0 THEN
		(* Write CSV header *)
		s1:='Title1;Title2,...';
		SysFileWrite(hFile, ADR(s1), LEN(s1));
		SysFileWrite(hFile, ADR(Logger_CRLF), LEN(Logger_CRLF));	(* End of line encoding	*)
	END_IF
ELSE
	(*** File exist *** Close file and reopen in append mode *)
	SysFileClose(hFile);
	hFile:=SysFileOpen(LogFileName,'a');
END_IF

(* Log to file *)
IF hFile<>0 THEN
	(* Date stamp *)
	s1:=REPLACE( Sys.Time_LogString , ' ' , 1 , 11 );
	SysFileWrite(hFile, ADR(s1), LEN(s1));
	(* Write CSV data *)
	s1:=CONCAT(';', 'Data1' );
	s1:=CONCAT(s1 , ';');
	s1:=CONCAT(s1 , 'Data2' );
	s1:=CONCAT(s1 , ';');
	s1:=CONCAT(s1 , '...' );
	SysFileWrite(hFile, ADR(s1), LEN(s1));
	(* Add line CRLF and close *)
	SysFileWrite(hFile, ADR(Logger_CRLF), LEN(Logger_CRLF));
	SysFileClose(hFile);
END_IF
END_FUNCTION

(* POU ClevergyUtils/FIND_OCCURRENCE, ST *)
FUNCTION FIND_OCCURRENCE : INT
VAR_INPUT
	SOURCE: STRING;
	TO_SEARCH: STRING;
	OCCURRENCE: INT;
END_VAR
VAR
	i:INT;
	tmp:STRING;
	cont:INT:=0;
END_VAR
cont:=0;
TMP:=SOURCE;

WHILE(LEN(TMP)>0) DO

	i:=FIND(SOURCE, TO_SEARCH);
	IF (i>0) THEN
		CONT:=CONT+1;
		TMP:=DELETE(SOURCE, i ,1);
		IF(cont=OCCURRENCE) THEN
			FIND_OCCURRENCE:=i;
			RETURN;
		END_IF
	END_IF

END_WHILE

FIND_OCCURRENCE:=0;

RETURN;
END_FUNCTION

(* POU ClevergyUtils/FLT_EVENT, ST *)
FUNCTION_BLOCK FLT_EVENT
VAR_INPUT
	IN		: BOOL;
	INITEV	: BOOL:=TRUE;
END_VAR
VAR_OUTPUT
	EVH		: BOOL;
	EVL		: BOOL;
END_VAR
VAR
	init	: BOOL:=FALSE;
	old		: BOOL;
END_VAR
EVH:=FALSE;
EVL:=FALSE;

IF NOT init THEN
	init:=TRUE;
	IF INITEV THEN
		old := NOT IN;
	ELSE
		old := IN;
	END_IF
END_IF

IF old<>IN THEN
	old:=IN;
	IF IN THEN EVH:=TRUE; ELSE EVL:=TRUE; END_IF
END_IF

(* NB: Questo functional block segnala l'EVENTO, NON lo STATO.
	   Infatti se IN non muta lo stato, sia EVL sia EVH rimangono FALSE *)
END_FUNCTION_BLOCK

(* POU ClevergyUtils/FLT_KEY, ST *)
FUNCTION_BLOCK FLT_KEY
VAR_INPUT
	IN		: BOOL;
	TTAP	: TIME:=T#5s;
	INITEV	: BOOL:=TRUE;
END_VAR
VAR_OUTPUT
	OUT		: BOOL;
	EVH		: BOOL;
	EVL		: BOOL;
END_VAR
VAR
	init	: BOOL:=FALSE;
	timer	: TON;
	timerIn	: TON;				(* Inhibition timer *)
	fInhibit: BOOL:=FALSE;
END_VAR
EVH:=FALSE;
EVL:=FALSE;

IF NOT init THEN
	init := TRUE;
	IF INITEV THEN
		OUT  := NOT IN;
	ELSE
		OUT  := IN;
	END_IF
END_IF

timerIn(IN:=fInhibit,PT:=T#500ms);

IF timerIn.Q THEN fInhibit := FALSE; END_IF

IF NOT fInhibit THEN

	IF OUT<>IN THEN
		timer(IN:=TRUE,PT:=TTAP);
		IF timer.Q THEN
			OUT:=IN;
			timer(IN:=FALSE);
			fInhibit := TRUE;
			IF OUT THEN EVH:=TRUE; ELSE EVL:=TRUE; END_IF
		END_IF
	ELSE
		timer(IN:=FALSE);
	END_IF
END_IF
END_FUNCTION_BLOCK

(* POU ClevergyUtils/FLT_TIME, ST *)
FUNCTION_BLOCK FLT_TIME
VAR_INPUT
	IN		: BOOL;
	TTAP	: TIME:=T#5s;
	INITEV	: BOOL:=TRUE;
END_VAR
VAR_OUTPUT
	OUT		: BOOL;
	EVH		: BOOL;
	EVL		: BOOL;
END_VAR
VAR
	init	: BOOL:=FALSE;
	timer	: TON;
END_VAR
EVH:=FALSE;
EVL:=FALSE;

IF NOT init THEN
	init := TRUE;
	IF INITEV THEN
		OUT  := NOT IN;
	ELSE
		OUT  := IN;
	END_IF
END_IF

IF OUT<>IN THEN
	timer(IN:=TRUE,PT:=TTAP);
	IF timer.Q THEN
		OUT:=IN;
		timer(IN:=FALSE);
		IF OUT THEN EVH:=TRUE; ELSE EVL:=TRUE; END_IF
	END_IF
ELSE
	timer(IN:=FALSE);
END_IF
END_FUNCTION_BLOCK

(* POU GeoLumenWrapping/GeolumenNodeList, ST *)
FUNCTION_BLOCK GeolumenNodeList (*Esegue la lettura dei mac address e del numero id associato nel file x_Lux_List.txt dove x è il numero id del plc*)
VAR_OUTPUT
	Message		: STRING;
END_VAR
VAR CONSTANT
	RTS_INVALID_HANDLE : DWORD:=0;
	AM_READ: STRING [20]:= 'r';			(* Use 'w' (write), 'r' (read) or 'rw' (read and write) *)
	MAX_LINE_CHARLEN:WORD:=100;
END_VAR
VAR
	(*hMode		: ACCESS_MODE;
	hFile		: RTS_IEC_HANDLE;
	hRes		: RTS_IEC_RESULT;  *)
	bList		: ARRAY [0..MAX_LINE_CHARLEN] OF BYTE;
	bListLen :INT;
	hFile		: DWORD;

	i, j			: DWORD;
	k, x			: INT;
	xwDimFile	: LWORD;
	bChar		: BYTE;
	sFileName 	: STRING;
	ValueToInsert: WORD;
	wLocal		: WORD;
	bIndex:INT;
	lastPosSeparator:INT;
	pot:WORD;
	xRel:INT;
END_VAR
Message:='';
bIndex:=0;
lastPosSeparator:=0;
pot:=0;
FOR i:=0 TO MAX_LINE_CHARLEN DO
	BList[i]:=0;
END_FOR
hfile:=0;
(* Open data file *)
sFileName:=CONCAT(STR1:=MapConf_Path, STR2:=PLC_ID);
sFileName:=CONCAT(STR1:=sFileName, STR2:=Luxlist_FileName);
hFile:=SysFileOpen(sFileName,AM_READ);

(* File not found *)
IF hFile=RTS_INVALID_HANDLE THEN
	Message:='File not found';
	RETURN;
END_IF

(* Close file *)
SysFileClose(hFile);

(* Open data file *)
i:=0;
j:=0;
k:=0;
x:=0;
bListLen:=0;
wLocal:=0;
ValueToInsert:=0;
bChar:=0;
xwDimFile:=0;
hFile:=SysFileOpen(sFileName,AM_READ);

SysFileSetPos(hFile, i);
SysFileRead(hFile, ADR(bList[j]), 1);

(* WHILE NOT (SysFileEOF(hFile)) DO  *)
REPEAT
	IF bList[j] = 16#2F  (* se trovo '/'  *)
		THEN
			SysFileSetPos(hFile, i+1);
			SysFileRead(hFile, ADR(bList[j+1]), 1);
			IF bList[j+1] = 16#2F (* se trovo ancora '/'  *)
				THEN
					WHILE  bList[j]<> 16#0D DO
						i := i+1;
						SysFileSetPos(hFile, i);	
						SysFileRead(hFile, ADR(bList[j]), 1);
					END_WHILE
					i := i+1;
					SysFileSetPos(hFile, i);
					SysFileRead(hFile, ADR(bList[j]), 1);
					IF bList[j] = 16#0A
						THEN 
							i := i+1;
							j := 0;
							SysFileSetPos(hFile, i);	
							SysFileRead(hFile, ADR(bList[j]), 1); (*leggo il primo carattere della nuova riga  *)
						ELSE
							Message:='Errore 0D 0A';
							RETURN;
					END_IF
				ELSE
					Message:='Errore //';
					RETURN;
			END_IF
	END_IF
	IF bList[j] <> 16#3B (*finchè non trovo ;   *)
		THEN
			IF bList[j] = 16#2C THEN
				lastPosSeparator:=DWORD_TO_INT(j);
			END_IF
			i:=i+1;
			j:=j+1;
			bListLen:=bListLen+1;
		ELSE
			i:=i+3;   (* Se trovo ; inizio a salvare i dati della riga letta in TabListLux[k]....  *)
			j:=0;
			k:=k+1;
			FOR bIndex:=0 TO lastPosSeparator-1 DO
				pot:=lastPosSeparator-1 -bIndex;
				TabListLux[k].LuxNumber :=TabListLux[k].LuxNumber+BYTE_TO_DWORD(bList[bIndex]-16#30)*REAL_TO_DWORD(EXPT(10,pot)) ;  (*   memorizzo il numero del lux   *)
			END_FOR
			TabListLux[k].StMacAdd:='';
			FOR x:=lastPosSeparator+1 TO bListLen-1 DO
				CASE bList[x] OF
					16#61: bList[x]:=16#41;
					16#62: bList[x]:=16#42;
					16#63: bList[x]:=16#43;
					16#64: bList[x]:=16#44;
					16#65: bList[x]:=16#45;
					16#66: bList[x]:=16#46;
				END_CASE
				TabListLux[k].StMacAdd:= CONCAT(TabListLux[k].StMacAdd, ASCIIBYTE_TO_STRING(bList[x]));
			END_FOR
			FOR x:=lastPosSeparator+1 TO lastPosSeparator+1+3  DO
				xRel:=x-(lastPosSeparator+1);
				 IF( bList[x]<=16#39 AND  bList[x]>=16#30)
				THEN
					wLocal:=BYTE_TO_WORD(bList[x]-16#30);
					TabListLux[k].MacAddH :=  TabListLux[k].MacAddH + SHL(wLocal, 12-(xRel)*4); (* Corrisponde a  4*(7-x)   *)
				ELSE

					CASE  bList[x] OF
						16#61, 16#41:
							ValueToInsert:= 16#0A;
							TabListLux[k].MacAddH :=  TabListLux[k].MacAddH + SHL( ValueToInsert, 12-(xRel)*4);
						16#62, 16#42:
							ValueToInsert:= 16#0B;
							TabListLux[k].MacAddH :=  TabListLux[k].MacAddH + SHL( ValueToInsert, 12-(xRel)*4);
						16#63, 16#43:
							ValueToInsert:= 16#0C;
							TabListLux[k].MacAddH :=  TabListLux[k].MacAddH + SHL( ValueToInsert, 12-(xRel)*4);
						16#64, 16#44:
							ValueToInsert:= 16#0D;
							TabListLux[k].MacAddH :=  TabListLux[k].MacAddH + SHL( ValueToInsert, 12-(xRel)*4);
						16#65, 16#45:
							ValueToInsert:= 16#0E;
							TabListLux[k].MacAddH :=  TabListLux[k].MacAddH + SHL( ValueToInsert, 12-(xRel)*4);
						16#66, 16#46:
							ValueToInsert:= 16#0F;
							TabListLux[k].MacAddH :=  TabListLux[k].MacAddH + SHL( ValueToInsert, 12-(xRel)*4);
					END_CASE
				END_IF
			END_FOR
			FOR x:=lastPosSeparator+1+4 TO lastPosSeparator+1+4+3 DO
				xRel:=x-(lastPosSeparator+1+4);
				 IF( bList[x]<=16#39 AND  bList[x]>=16#30)
				THEN
					wLocal:=BYTE_TO_WORD(bList[x]-16#30);
					TabListLux[k].MacAddL :=  TabListLux[k].MacAddL + SHL(wLocal, 12-(xRel)*4); (* Corrisponde a  4*(7-x)   *)
				ELSE

					CASE  bList[x] OF
						16#61, 16#41:
							ValueToInsert:= 16#0A;
							TabListLux[k].MacAddL :=  TabListLux[k].MacAddL + SHL( ValueToInsert, 12-(xRel)*4);
						16#62, 16#42:
							ValueToInsert:= 16#0B;
							TabListLux[k].MacAddL :=  TabListLux[k].MacAddL + SHL( ValueToInsert, 12-(xRel)*4);
						16#63, 16#43:
							ValueToInsert:= 16#0C;
							TabListLux[k].MacAddL :=  TabListLux[k].MacAddL + SHL( ValueToInsert, 12-(xRel)*4);
						16#64, 16#44:
							ValueToInsert:= 16#0D;
							TabListLux[k].MacAddL :=  TabListLux[k].MacAddL + SHL( ValueToInsert, 12-(xRel)*4);
						16#65, 16#45:
							ValueToInsert:= 16#0E;
							TabListLux[k].MacAddL :=  TabListLux[k].MacAddL + SHL( ValueToInsert, 12-(xRel)*4);
						16#66, 16#46:
							ValueToInsert:= 16#0F;
							TabListLux[k].MacAddL :=  TabListLux[k].MacAddL + SHL( ValueToInsert, 12-(xRel)*4);
					END_CASE
				END_IF
			END_FOR
			TabListLux[k].MacAdd:=SHL(TabListLux[k].MacAddH, 16)+TabListLux[k].MacAddL;
			bListLen:=0;
			lastPosSeparator:=0;
			pot:=0;
	END_IF
	SysFileSetPos(hFile, i);
	SysFileRead(hFile, ADR(bList[j]), 1);
UNTIL  ((SysFileEOF(hFile)) AND ( bList[j] <> 16#3B))
END_REPEAT
(* END_WHILE  *)
IF SysFileEOF(hFile) = 0
	THEN Message:='Reading Default_Lux File: OK';
END_IF

(* Close file *)
SysFileClose(hFile);
END_FUNCTION_BLOCK

(* POU ClevergyUtils/Utils Functions/GETBIT, ST *)
FUNCTION GETBIT : BOOL
VAR_INPUT
		IN		:	DWORD;
		Offset	:	BYTE;
END_VAR
VAR
END_VAR
GETBIT := DWORD_TO_BOOL(IN AND(SHL(DWORD#1,Offset)));
END_FUNCTION

(* POU GeoLumenWrapping/getGeolumenIDbyLuxID, ST *)
FUNCTION getGeolumenIDbyLuxID : DWORD
VAR_INPUT
	LuxID:WORD;
END_VAR
VAR
	i:INT;
END_VAR
IF LuxID = 0 THEN
	getGeolumenIDbyLuxID:=0;
END_IF
FOR i:=1 TO MAX_LUXNUM DO
	IF TabListLux[i].LuxNumber=LuxID THEN
		getGeolumenIDbyLuxID:=TabListLux[i].LuxID_Geolumen;
		RETURN;
	END_IF
END_FOR
END_FUNCTION

(* POU GeoLumenWrapping/getGeolumenNodeByLuxId, ST *)
FUNCTION getGeolumenNodeByLuxId : INT
VAR_INPUT
	LuxID : INT;
END_VAR

VAR
	I : INT;
END_VAR
getGeolumenNodeByLuxId:=-1;
FOR I:=1 TO MAX_LUXNUM DO
	IF (LuxGeolumenNodes[i].ID_Lux = LuxID) THEN getGeolumenNodeByLuxId :=i; RETURN; END_IF
END_FOR
END_FUNCTION

(* POU GeoLumenWrapping/getLuxIDbyGeolumenID, ST *)
FUNCTION getLuxIDbyGeolumenID : DWORD
VAR_INPUT
	GeolumenID:WORD;
END_VAR
VAR
	i:INT;
END_VAR
IF GeolumenID = 0 THEN
	getLuxIDbyGeolumenID:=0;
	RETURN;
END_IF
getLuxIDbyGeolumenID:=0;
FOR i:=1 TO MAX_LUXNUM DO
	IF TabListLux[i].LuxID_Geolumen=GeolumenID THEN
		getLuxIDbyGeolumenID:=TabListLux[i].LuxNumber;
		RETURN;
	END_IF
END_FOR
END_FUNCTION

(* POU ClevergyUtils/Intero_WORD, ST *)
FUNCTION Intero_WORD : WORD
VAR_INPUT
	IN_INT: INT;
END_VAR
VAR
	Appoggio:DINT;
END_VAR
IF IN_INT<0 THEN
	Appoggio:= (65534 + IN_INT);
	Intero_WORD:= (DINT_TO_WORD(Appoggio));
ELSE
	Intero_WORD:= INT_TO_WORD(IN_INT);
END_IF
END_FUNCTION

(* POU ClevergyUtils/IS_DST, ST *)
FUNCTION IS_DST : BOOL
VAR_INPUT
	countryCode : STRING;
END_VAR
VAR
	tmp:DATE;
	i:DINT;
	iDW:UINT;
	lastSunday:DINT;
	localTime:DT;
	currDate:DATE;
	currMonth:INT;
	currDay:DINT;
	currDayOfWeek:INT;
	currHour:INT;
END_VAR
IS_DST:=FALSE;

localTime:=SysRtcGetTime(TRUE);
currDate:=DT_TO_DATE(localTime);
currDay:=DAY_OF_DATE(currDate);
currDayOfWeek:=DAY_OF_WEEK(currDate);
currMonth:=MONTH_OF_DATE(currDate);
currHour:=HOUR_OF_DT(localTime);

IF countryCode = 'IT' THEN

	(* data corrente tra Aprile e Ottobre => DST true *)
	IF(currMonth> 3 AND currMonth < 10) THEN IS_DST:=TRUE; RETURN; END_IF

	IF(currMonth < 3 OR currMonth > 10) THEN IS_DST:=FALSE; RETURN; END_IF

	(* è Marzo *)
	IF(currMonth= 3) THEN
		lastSunday:=0;  (* init a 0, per caso in cui il giorno corrente è già oltre l'ultima domenica del mese*)
		iDW:=currDayOfWeek;
		FOR i:= currDay TO 31 DO
			IF(iDW=7) THEN lastSunday:=i; END_IF
			iDW:=((iDW+1) MOD 8)+iDW/8;
		END_FOR
		IF(currDay > lastSunday OR ( currDay = lastSunday AND currHour>=2)) THEN
			IS_DST:=TRUE; RETURN;
		ELSE
			IS_DST:=FALSE; RETURN;
	 	END_IF
	END_IF

	(* è Ottobre *)
	IF(currMonth= 10) THEN
		iDW:=currDayOfWeek;
		lastSunday:=0; (* init a 0, per caso in cui il giorno corrente è già oltre l'ultima domenica del mese*)
		FOR i:=currDay TO 31 DO
			IF(iDW=7) THEN lastSunday:=i; END_IF
			iDW:=((iDW+1) MOD 8)+iDW/8;
		END_FOR
		IF(currDay <lastSunday OR ( currDay=lastSunday AND currHour<=2)) THEN
			IS_DST:=TRUE; RETURN;
		ELSE
			IS_DST:=FALSE; RETURN;
	 	END_IF
	END_IF


END_IF
END_FUNCTION

(* POU ClevergyUtils/LAMP_AL_GENERALE, ST *)
FUNCTION_BLOCK LAMP_AL_GENERALE
VAR_INPUT

	Allarme: BOOL;
	Warning: BOOL;
END_VAR
VAR_OUTPUT
	StatoSistema:BYTE;
	SistemaInAllarme:BOOL;
	SistemaWarning:BOOL;
	AllarmeLampada:BOOL;
END_VAR
VAR
	Lampeggio:BLINK;
END_VAR
IF Allarme THEN       					(* Se Allarme Attivo Luce fissa ON *)
	StatoSistema:=2;
	SistemaInAllarme:=TRUE;
	SistemaWarning:=FALSE;
	AllarmeLampada:=TRUE;
ELSIF Warning THEN					(* Se Allarme Attivo Luce fissa pulse *)
	StatoSistema:=1;
	SistemaInAllarme:=FALSE;
	SistemaWarning:=TRUE;
	Lampeggio(ENABLE:=TRUE , TIMELOW:=t#1s , TIMEHIGH:=t#1s , OUT=>AllarmeLampada );
ELSE
	StatoSistema:=0;
	SistemaInAllarme:=FALSE;
	SistemaWarning:=FALSE;
	AllarmeLampada:=FALSE;
END_IF
END_FUNCTION_BLOCK

(* POU ClevergyUtils/Utils Functions/LINEAR, ST *)
FUNCTION LINEAR : REAL (* Linear interpolation *)
VAR_INPUT
	X_In	: REAL;
	P1_X	: REAL;
	P1_Y	: REAL;
	P2_X	: REAL;
	P2_Y	: REAL;
END_VAR
VAR
END_VAR
LINEAR:=P1_Y+(((P2_Y-P1_Y)*(X_In-P1_X))/(P2_X-P1_X));
END_FUNCTION

(* POU ClevergyUtils/Utils Functions/LINEAR_BAD, ST *)
FUNCTION LINEAR_BAD : INT (* Linear interpolation *)
VAR_INPUT
	PuntoMinX	: INT;
	PuntoMaxX	: INT;
	ValIn		: INT;
	PuntoMinY	: REAL;
	PuntoMaxY	: REAL;
	Decimali	: BYTE;
END_VAR
VAR
	Gain				: REAL;
	PuntoMinX_R			: REAL;
	PuntoMaxX_R			: REAL;
	Linearizzazione_R	: REAL;
END_VAR
PuntoMinX_R:=INT_TO_REAL(PuntoMinX);
PuntoMaxX_R:=INT_TO_REAL(PuntoMaxX);

Gain:=(PuntoMaxX_R-PuntoMinX_R)/(PuntoMaxY-PuntoMinY);	(* Calcolo in guadagno per la linarizzazione *)
Linearizzazione_R:=PuntoMinx+(Gain*(ValIn-PuntoMinY));	(* Ottengo il valore linearizzato *)

LINEAR_BAD:=REAL_TO_INT(Linearizzazione_R*(EXPT(10, Decimali)));  (* Ottengo intero con i decimai voluti *)
END_FUNCTION

(* POU GeoLumenWrapping/Debug/logRequestSTS0, ST *)
FUNCTION logRequestSTS0 : BOOL
VAR_INPUT
	message:STRING(255);
END_VAR
VAR
	hName : STRING(255) :='REQUEST_STS0.TXT';
	hFile	 : DWORD;
	tmp:STRING(255);
END_VAR
tmp:=CONCAT(DWORD_TO_STRING(Plant_SN),'_');
hName:=CONCAT(tmp,hName);
hName:=CONCAT(FilesPath ,hName);
hFile:=SysFileOpen(hName,'a');
IF hFile<>0 THEN

	tmp:=DT_TO_STRING(SYS.Time_CT_DT);
	SysFileWrite(hFile, ADR(TMP),LEN(TMP));
	SysFileWrite(hFile, ADR(message),LEN(message));
	tmp:='$R$N';
	SysFileWrite(hFile, ADR(TMP),LEN(TMP));
	SysFileClose(hFile);

END_IF
END_FUNCTION

(* POU GeoLumenWrapping/Debug/logSerialInMessage, ST *)
FUNCTION logSerialInMessage : BOOL
VAR_INPUT
	message:STRING(255);
END_VAR
VAR
	hName : STRING(255) :='DEBUG_SERIAL.TXT';
	hFile	 : DWORD;
	tmp:STRING(255);
END_VAR
hName:=CONCAT(FilesPath ,hName);
hFile:=SysFileOpen(hName,'a');
IF hFile<>0 THEN

	tmp:=DT_TO_STRING(SYS.Time_CT_DT);
	SysFileWrite(hFile, ADR(TMP),LEN(TMP));
	SysFileWrite(hFile, ADR(message),LEN(message));
	tmp:='$R$N';
	SysFileWrite(hFile, ADR(TMP),LEN(TMP));
	SysFileClose(hFile);

END_IF
END_FUNCTION

(* POU GeoLumenWrapping/Debug/logSerialInMessageRaw, ST *)
FUNCTION logSerialInMessageRaw : BOOL
VAR_INPUT
	message:STRING(255);
END_VAR
VAR
	hName : STRING(255) :='DEBUG_SERIAL_RAW.TXT';
	hFile	 : DWORD;
	tmp:STRING(255);
END_VAR
tmp:=CONCAT(DWORD_TO_STRING(Plant_SN),'_');
tmp:=CONCAT(tmp, WORD_TO_STRING(SYS.Time_Year));
tmp:=CONCAT(tmp, WORD_TO_STRING(SYS.Time_Month));
tmp:=CONCAT(tmp, WORD_TO_STRING(SYS.Time_Day));
tmp:=CONCAT(tmp, '_');
hName:=CONCAT(tmp,hName);
hName:=CONCAT(FilesPath ,hName);
hFile:=SysFileOpen(hName,'a');
IF hFile<>0 THEN

	SysFileWrite(hFile, ADR(message),LEN(message));
	SysFileClose(hFile);

END_IF
END_FUNCTION

(* POU ClevergyUtils/MEAN_VALUE, ST *)
FUNCTION MEAN_VALUE : WORD
VAR_INPUT
		pArray	:	POINTER TO ARRAY [1..2] OF WORD;
		Length	:	WORD;
END_VAR
VAR
		counter	:	WORD;
		Sum		:	DWORD;
		(*Maximum	:	WORD;
		Minimum	:	WORD;*)
END_VAR
Sum := 0;
(*Maximum := 0;
Minimum := 0;*)

FOR counter:=1 TO Length BY 1 DO
	Sum := Sum + WORD_TO_DWORD(pArray^[counter]);

	(*IF pArray^[counter] > Maximum THEN Maximum := pArray^[counter]; END_IF
	IF pArray^[counter] < Minimum THEN Minimum := pArray^[counter]; END_IF*)

END_FOR

(*Sum := Sum - WORD_TO_DWORD(Maximum) - WORD_TO_DWORD(Minimum);
MEAN_VALUE := DWORD_TO_WORD(Sum/(Length-2));*)

MEAN_VALUE := DWORD_TO_WORD(Sum/Length);
END_FUNCTION

(* POU ClevergyUtils/MEAN_VALUE_dint, ST *)
FUNCTION MEAN_VALUE_dint : DINT
VAR_INPUT
		pArray	:	ARRAY [1..200] OF DINT;
		Length	:	WORD;
END_VAR
VAR
		counter	:	WORD;
		Sum		:	DINT;
		(*Maximum	:	WORD;
		Minimum	:	WORD;*)
END_VAR
Sum := 0;
(*Maximum := 0;
Minimum := 0;*)

FOR counter:=1 TO Length BY 1 DO
	Sum := Sum + pArray[counter];

	(*IF pArray^[counter] > Maximum THEN Maximum := pArray^[counter]; END_IF
	IF pArray^[counter] < Minimum THEN Minimum := pArray^[counter]; END_IF*)

END_FOR

(*Sum := Sum - WORD_TO_DWORD(Maximum) - WORD_TO_DWORD(Minimum);
MEAN_VALUE := DWORD_TO_WORD(Sum/(Length-2));*)

MEAN_VALUE_dint := Sum/Length;
END_FUNCTION

(* POU ClevergyUtils/MEMCLR, ST *)
FUNCTION MEMCLR:BOOL
VAR_INPUT
	pDestinationAddress:POINTER TO ARRAY[1..2] OF BYTE;
	BytesToClear:WORD;
END_VAR
VAR
END_VAR
WHILE (BytesToClear > 0) DO
	pDestinationAddress^[1]:=0;
	pDestinationAddress:=ADR(pDestinationAddress^[2]); (* increment destination *)
	BytesToClear:=BytesToClear -1; (* decrement number of bytes to copy *)
END_WHILE
END_FUNCTION

(* POU obj_ASTR, ST *)
FUNCTION_BLOCK obj_ASTR
(* === Block for realizing the ASTR block ===
	
	The ASTR is a CRON-like block  whose setpoint is determined by  the assigned schedule AND the times of sunrise and sunset.
   	
	Versioning:
		v1.0 [18/03/16] - Diego Bernini
*)

VAR_INPUT
	(* Logical ID of the ASTRO CRON, univocal w.r.t the plant *)
	ID : DWORD;

	(* the local time, provided by the local RTC *)
	localTime :DT;

	(* time offsett of the local timew.r.t. UTC time: +/- hours - DO NOT COUNT DST WHICH IS AUTOMALLY CALCULATED*)
	rOffsetToUTC :REAL:=1;

	(* code of the country for enabling the autodetection of DaylightSaving *)
	(* currently only Italy is supported *)
	countryCode :STRING(25);
	(*latitude *)
	rLatitude : REAL:=45.660952;
	(*longitude *)
	rLongitude : REAL:=9.652085;

END_VAR

VAR_INPUT

	(*twilight morning mode, 0-100
	    it determines how the civil sunrise is exploited (sun at -6° below the horizon).	
	     0 => morning twilight is not exploited, hence official sunrise time is calculated
	     100 => morning twilight is fully exploited, hence official sunrise time is calculated
                0<mode<100 intermediate valutes
	*)
	twilightMorningMode : BYTE:=0;

	(*twilight evening mode, 0-100
	    it determines how the civil sunset is exploited (sun at -6° below the horizon).	
	     0 => evening twilight is not exploited, hence official sunset time is calculated
	     100 => evening twilight is fully exploited, hence official sunset time is calculated
                0<mode<100 intermediate valutes
	*)
	twilightEveningMode : BYTE:=0;

	(* parameters for adjusting the computed times of sunsent and sunrise *)
	preSunset : BYTE:=0;
	postSunset:  BYTE:=0;

	preSunrise:BYTE:=0;
	postSunrise:BYTE:=0;
END_VAR
VAR_OUTPUT
	(* the setPoint, computer considering both the CRON scheduling and the [sunset, sunrise] interval *)
	setPoint : INT;
	(* the times of sunset and sunrise *)
	dtSunriseOfficial : DT;
	dtSunsetOfficial : DT;
	dtSunriseCivilTwilight : DT;
	dtSunsetCivilTwilight  : DT;
END_VAR
VAR

	init: BOOL:=FALSE;
	myCRON : obj_CRON;
	(* variables for astro calculations *)
	dtUTC_Time :DT;
	myTimeZone :REAL;
	bDaylightSavingActive : BOOL;
	timeStart: DT;
	timeEnd: DT;
	status :BYTE  :=0;
	localCorrection : TIME;

	obJAstroOscat : SUN_TIME;
	currentDateUCT : DATE;

	extensionTwilightEvening : TIME;
	advanceTwilightMorning : TIME;
	localDate:DATE;
	oldDate:DATE;


END_VAR
(* init the object *)
astroInit();

(* update the internal CRON *)
myCron();

(* obtaining the local Date *)
localDate:=DT_TO_DATE(localTime);

(* sunrise and sunset time could be calcualted only when the date change --disabled now*)
(* IF(oldDate <> localDate) THEN *)

	oldDate:=localDate;

	(* computing the difference from local time  w.r.t. UTC time *)
	localCorrection:=REAL_TO_TIME(myTimeZone);
	bDaylightSavingActive:=IS_DST(countryCode);
	IF bDaylightSavingActive  THEN localCorrection:=localCorrection + T#1h; END_IF

	(* obtain UTC time, for check *)
	dtUTC_Time:=localTime-localCorrection;

	(* calculating official sunrise and sunse times *)
	obJAstroOscat(h:=-0.83333, (* -0.83333° instead of 0°, for correcting the refraction at horizon *)
			UTC:=localDate,
			Latitude:=rLATITUDE,
			Longitude:=rLONGITUDE);

	(* notice: the values calcualted by the OSCAT object are in UTC time, so we need to sum the localCorrection *)
	dtSunriseOfficial:=DWORD_TO_DT(DATE_TO_DWORD(localDate)+(TOD_TO_DWORD(obJAstroOscat.SUN_RISE)/1000))+localCorrection;
	dtSunsetOfficial:=DWORD_TO_DT(DATE_TO_DWORD(localDate)+(TOD_TO_DWORD(obJAstroOscat.SUN_SET)/1000))+localCorrection;

	(* calculating civil twilight times *)
	obJAstroOscat(h:=-6, (* -6° civil twilight horizon *)
			UTC:=localDate,
			Latitude:=rLATITUDE,
			Longitude:=rLONGITUDE);

	dtSunriseCivilTwilight:=DWORD_TO_DT(DATE_TO_DWORD(localDate)+(TOD_TO_DWORD(obJAstroOscat.SUN_RISE)/1000))+localCorrection;
	dtSunsetCivilTwilight:=DWORD_TO_DT(DATE_TO_DWORD(localDate)+(TOD_TO_DWORD(obJAstroOscat.SUN_SET)/1000))+localCorrection;

(*END_IF*)

(* now the duration of twilights are computed and scaled according to the mode percentage, *)
(* in order to obtain the extensions to sum to the official times *)

extensionTwilightEvening:=REAL_TO_TIME(TIME_TO_REAL(dtSunsetCivilTwilight-dtSunsetOfficial)*(BYTE_TO_REAL(twilightEveningMode)/100));
advanceTwilightMorning:=REAL_TO_TIME(TIME_TO_REAL(dtSunriseOfficial-dtSunriseCivilTwilight)*(BYTE_TO_REAL(twilightMorningMode)/100));

timeStart:=dtSunsetOfficial+extensionTwilightEvening;
timeEnd:= dtSunriseOfficial-advanceTwilightMorning;

(* apply the corrections *)

IF(preSunrise <> 0) THEN
	timeEnd:= timeEnd - DWORD_TO_TIME(preSunrise*1000*60);
ELSIF (postSunrise<>0) THEN
	timeEnd:= timeEnd +  DWORD_TO_TIME(postSunrise*1000*60);
END_IF

IF(preSunset <> 0) THEN
	timeStart:= timeStart - DWORD_TO_TIME(preSunset*1000*60);
ELSIF (postSunset<>0) THEN
	timeStart:= timeStart +  DWORD_TO_TIME(postSunset*1000*60);
END_IF


(* return the setPoint:
     - if localTime inside [timeStart, timeEnd] => crono setPoint
     - 0 otherwise
*)

IF (localTime>=timeStart OR  localTime<=timeEnd) THEN


	SetPoint:=myCron.SetPoint;

ELSE
	SetPoint:=0;

END_IF
END_FUNCTION_BLOCK
ACTION AddLogData:
Logger.s1:=INSERT('&ASTR=',DWORD_TO_STRING(ID),5);
IF ID<10 THEN Logger.s1:=INSERT(Logger.s1,'0',5); END_IF

Logger.s1:=CONCAT(Logger.s1,INT_TO_STRING(SetPoint));														Logger.s1:=CONCAT(Logger.s1,';');

Logger.s1:=CONCAT(Logger.s1,BYTE_TO_STRING(Status));														Logger.s1:=CONCAT(Logger.s1,';');

Logger.s1:=CONCAT(Logger.s1,BYTE_TO_STRING(twilightEveningMode));											Logger.s1:=CONCAT(Logger.s1,';');

(* iso format *)
Logger.s1:=CONCAT(Logger.s1,REPLACE(DELETE(DT_TO_STRING(dtSunriseOfficial), LEN:=3, POS:=1), 'T', 1, 11));			Logger.s1:=CONCAT(Logger.s1,';');

Logger.s1:=CONCAT(Logger.s1,REPLACE(DELETE(DT_TO_STRING(dtSunsetOfficial), LEN:=3, POS:=1), 'T', 1, 11));				Logger.s1:=CONCAT(Logger.s1,';');

Logger.s1:=CONCAT(Logger.s1,REPLACE(DELETE(DT_TO_STRING(dtSunriseCivilTwilight), LEN:=3, POS:=1), 'T', 1, 11));			Logger.s1:=CONCAT(Logger.s1,';');

Logger.s1:=CONCAT(Logger.s1,REPLACE(DELETE(DT_TO_STRING(dtSunsetCivilTwilight), LEN:=3, POS:=1), 'T', 1, 11)); 			Logger.s1:=CONCAT(Logger.s1,';');

Logger.s1:=CONCAT(Logger.s1,BYTE_TO_STRING(twilightMorningMode));

ADDSTRING(ADR(Logger.TData), ADR(Logger.s1), Logger.TLen);
END_ACTION
ACTION astroInit:
IF(NOT init) THEN
	myCRON(ID:=ID,crono_type:='ASTR');
	myTimeZone:=rOffsetToUTC*1000*60*60; (* timezone in millseconds *)
	init := TRUE;
END_IF
END_ACTION
ACTION restartInternalCrono:
init:=FALSE;
myCRON.InitOK:=FALSE;
END_ACTION

(* POU Plant_Objects/obj_CRON, ST *)
FUNCTION_BLOCK obj_CRON
(* === CRONOGRAFO STANDARD ===
   v1.0[16/04/15] - Versioning
   v1.1[19/05/15] - Removed DB creation from previous year
*)
VAR_INPUT
	CRONO_TYPE : STRING:='CR';
	(* Settings *)
	ID			: DWORD;		(* Index of instanced object *)

	InitOK		: BOOL;
	Alarm		: BOOL;
	Warning		: BOOL;

	Profile		: typ_Cron_Profile; 				(* Profilo attivo *)
	ProfileNr	: BYTE;								(* Indice profilo attivo *)
	CalendarIdx : WORD;								(* Indice calendario attivo *)
	Jolly		: ARRAY[0..9] OF typ_Cron_Jolly;	(* Jolly attivi *)

END_VAR
VAR_IN_OUT
END_VAR
VAR_OUTPUT
	SetPoint		: INT;
	(* Status *)
	Status_Log		: BYTE;
	Status_Vis 		: DWORD;
END_VAR
VAR
	Buf: 	ARRAY[0..512] OF BYTE; (* AVOID THIS!! *)
	hFile: 	DWORD;
	sFile: 	STRING;
	sFile2: STRING;

	i:		WORD;
	t1:		DWORD;
	t2:		BOOL;

END_VAR
VAR CONSTANT

	COLOR_RED			: DWORD	:= 16#2020F0;
	COLOR_YELLOW		: DWORD	:= 16#20F0F0;
	COLOR_GREEN			: DWORD	:= 16#20F020;
	COLOR_GREEN_OFF		: DWORD := 16#006000;
END_VAR
(* Check initialization *)
IF NOT InitOK THEN Init(); END_IF

(* Chrono *)
IF CalendarIdx<>Sys.Time_CT_Day THEN DB_Load(); END_IF
SetPoint:=Profile.Setpoint[Sys.Time_CT_Quarter];

(* Check jolly *)
FOR i := 0 TO 9 DO
	IF ( DT_TO_DWORD(Jolly[i].Start)>0  AND Jolly[i].End>Jolly[i].Start AND
	     Jolly[i].Start<=Sys.Time_CT_DT AND Jolly[i].End>Sys.Time_CT_DT ) THEN
			SetPoint:=Jolly[i].Temp;
	END_IF
END_FOR


(* Status color *)
   IF Alarm   THEN Status_Log:=2; Status_Vis:=COLOR_RED;
ELSIF Warning THEN Status_Log:=1; Status_Vis:=COLOR_YELLOW;
              ELSE Status_Log:=0; Status_Vis:=COLOR_GREEN;
			  END_IF
END_FUNCTION_BLOCK
ACTION DB_Create:
(*
Check presence of previous year *)
sFile2:=REPLACE(STR1:=sFile, STR2:=WORD_TO_STRING(Sys.Time_Year-1), L:=4, P:=LEN(FilesPath)+1);
hFile:=SysFileOpen(FileName:=sFile2, Mode:='r');
IF hFile<>0 THEN
	(* Check file version and close *)
	SysFileRead(File:=hFile, Buffer:=ADR(Buf), Size:=1);
	SysFileClose(File:=hFile);
END_IF
IF hFile<>0 AND Buf[0]=1 THEN
	(* Copy file *)
	SysFileCopy(FileDest:=sFile, FileSource:=sFile2);
ELSE

	(* Create empty file *)
	hFile:=SysFileOpen(FileName:=sFile, Mode:='w');

	MEMCLR(pDestinationAddress:=ADR(Buf), BytesToClear:=SIZEOF(Buf));
	FOR i := 0 TO 10239 BY 512 DO
		t1:=SysFileWrite(File:=hFile, Buffer:=ADR(Buf), Size:=512);
	END_FOR
	Buf[0]:=1;
	t2:=SysFileSetPos(File:=hFile, Pos:=0);
	t1:=SysFileWrite(File:=hFile, Buffer:=ADR(Buf), Size:=1);
	SysFileClose(File:=hFile);

END_IF
END_ACTION
ACTION DB_Load:
DB_SetName();

(* Open data file *)
hFile:=SysFileOpen(FileName:=sFile, Mode:='r');

(* File not found *)
IF hFile=0 THEN
	Warning:=TRUE;
	LogEv(EL_Wrn,EO_CRON,ID,1,'No_data_file');
	DB_Create();
	(* Reopen file *)
	hFile:=SysFileOpen(FileName:=sFile, Mode:='r');
	IF hfile=0 THEN
		Alarm:=TRUE;
		LogEv(EL_Alarm,EO_CRON,ID,3,'Filesystem_error');
		RETURN;
	END_IF
END_IF

(* Check version *)
SysFileRead(File:=hFile, Buffer:=ADR(Buf), Size:=1);
IF Buf[0]<>1 THEN
	IF NOT Alarm THEN
		Alarm:=TRUE;
		LogEv(EL_Alarm,EO_CRON,ID,2,'Bad_data_version');
	END_IF
	SysFileClose(File:=hFile);
	RETURN;
END_IF

(* Read Jolly data *)
t2:=SysFileSetPos(File:=hFile, Pos:=512);
t1:=SysFileRead(File:=hFile, Buffer:=ADR(Jolly), Size:=SIZEOF(Jolly));
(* Read active profile index *)
CalendarIdx:=Sys.Time_CT_Day;
t2:=SysFileSetPos(File:=hFile, Pos:=(1024+4*CalendarIdx));
t1:=SysFileRead(File:=hFile, Buffer:=ADR(ProfileNr), Size:=SIZEOF(ProfileNr));
(* Read active profile *)
t2:=SysFileSetPos(File:=hFile, Pos:=(3072+512*ProfileNr));
t1:=SysFileRead(File:=hFile, Buffer:=ADR(Profile), Size:=SIZEOF(Profile));

(* Close file and validate data *)
SysFileClose(File:=hFile);
END_ACTION
ACTION DB_SetName:
(* Create current filename 'yyyyCRnn.DAT' *)
sFile:=CONCAT(FilesPath,WORD_TO_STRING(Sys.Time_Year));
sFile:=CONCAT(STR1:=sFile, STR2:=CRONO_TYPE);
IF ID<10 THEN
sFile:=CONCAT(STR1:=sFile, STR2:='0');
END_IF
sFile:=CONCAT(STR1:=sFile, STR2:=DWORD_TO_STRING(ID));
sFile:=CONCAT(STR1:=sFile, STR2:='.DAT');
END_ACTION
ACTION Init:
DB_Load();
InitOK:=TRUE;
END_ACTION

(* POU GeoLumenWrapping/obj_GeolumenNode, ST *)
FUNCTION_BLOCK obj_GeolumenNode
VAR_INPUT
	(* ID del nodo, dal punto di vista delle rete - attenzione: cambia se alimentazione salta *)
	ID_Geolumen: DWORD;
	(*ID del LUX associato *)
	ID_LUX: DWORD;
	(*dimming desiderato *)
	desideredDimmValue:WORD;
	(*stato di feedback *)
	feedbackState: type_LuxGeolumenStatus;
	(*stato di echo comando *)
	echoCommandState: type_LuxGeolumenStatus;
	(*timestamp relativo all'ultima volta che si è ricevuto feedback di stato NEMAS dal nodo *)
	lastSeen:DT;
	(*timestamp relativo all'ultima volta che si è ricevuto feedback ECHO dal nodo *)
	echoLastSeen:DT;
	(*last parent*)
	lastPar:STRING;
	(*tempo oltre il quale il nodo viene ripingato *)
	MAX_NO_FEEDBACK_TIME:TIME:=t#5m; (*minutes*)
	MAX_NO_FEEDBACK_TIME_ABSOLUTE:TIME:=t#60m; (*minutes*)
	(*tentativi di ping raggiunti i quali il nodo viene considerato sparito *)
	MAX_RETRY_NO_FEEDBACK:WORD;
	(*tentativi di ping raggiunti i quali il nodo viene considerato con stato disallineato *)
	MAX_RETRY_STATUS_NOT_ALIGNED:WORD;
END_VAR
VAR_OUTPUT
	(*stato del nodo, secondo la nomenclatura Clevergy*)
	Status:BYTE;
	(*stato desiderato, costruito a partire dal desideredDimmValue *)
	desideredState: type_LuxGeolumenStatus;
	(*stringhe di get/set del nodo *)
	toSendSetString:STRING(255);
	GlobalMaxCurrent	: DWORD;
	GlobalMaxVoltage: DWORD;
	GlobalMaxPower: DWORD;
	toSendGetString:STRING(255);
	lampBroken:BOOL;
END_VAR
(*valori costanti dimmeraggio*)
VAR CONSTANT
	(*valori dimmeraggio min e max del nodo Geolumen*)
	MIN_DIMM:WORD:=0;
	MAX_DIMM:WORD:=1023;
	(*valore dimmeraggio max del LUX dal punto di vista della piattaforma Clevergy *)
	MAX_DIMM_LUX_CLEVERGY:WORD:=100;
END_VAR
VAR
	dayFeed:DWORD;
	(*var interne di appoggio *)
	fltNodeDisappeared:FLT_EVENT;
	retryDisappear:BYTE:=0;
	retryStatusNotAligned:BYTE:=0;
	timerAlive:TON;
	fltNodeStatusNotAligned:FLT_EVENT;
	timerAlignStatus:TON;
	templateDimm : STRING(255);
	templateGet : STRING(255);
	tmpNum:STRING(255);
	commandString:STRING(255);
	sendString:STRING(255);
	normalizedDesideredDimmValueGeoLumen:REAL;
	i:INT;
	fNormValue:WORD;
	fTemp1,fTemp2,fTemp3,fTemp4:REAL;
	tempConfronto:BOOL;
	tempConfrontoALive:TIME;
	tmpString:STRING(255);
	isBootedFlag:BOOL;
	tmpTime:TIME;
END_VAR
;
END_FUNCTION_BLOCK
ACTION checkAlive:
(*invia periodicamente re-get, per verificare nodo vivo*)
(*disabilitato per il momento*)

IF USING_EXTERNAL_ASTRO AND tmpBoolGoffDay THEN RETURN; END_IF

TimerAlive(IN:=NOT TimerAlive.Q,PT:=T#5m);
IF TimerAlive.Q THEN
	SendDataQueue(pTxData:=ADR(toSendGetString));
	SendDataQueue.addMessage();
	retryDisappear:=retryDisappear+1;
END_IF
END_ACTION
ACTION checkStatusANDPresence:
IF ID_Geolumen = 0 THEN RETURN; END_IF

(*SE IL NODO NON LO SENTO DAL TEMPO LIMITE E NON HO RAGGIUNTO IL LIMITE MASSIMO DI TENTATIVI => VERIFICO SE IL E' NODO VIVO *)
(* ORA DISABLED*)
IF(Sys.Time_CT_DT-lastSeen>MAX_NO_FEEDBACK_TIME) THEN
	checkAlive();
END_IF

(*GESTIONE LOG EV PER NODO SPARITO/RITORNATO *)
fltNodeDisappeared(IN:=((Sys.Time_CT_DT-lastSeen>MAX_NO_FEEDBACK_TIME) AND retryDisappear>=MAX_RETRY_NO_FEEDBACK) OR (Sys.Time_CT_DT-lastSeen>MAX_NO_FEEDBACK_TIME_ABSOLUTE));
IF fltNodeDisappeared.EVH THEN
	LogEv(EL_Alarm,EO_LUX,ID_Lux,12,'Geolumen node disappeared');
END_IF
IF fltNodeDisappeared.EVL THEN
	LogEv(EL_Log,EO_LUX,ID_Lux,13,'Geolumen node came back');
	retryDisappear:=0;
END_IF

(*SE IL NODO HA LA STATO DISALLINEATO E NON HO RAGGIUNTO NUMERO MASSIMO DI TENTATIVI => CERCO DI RIALLINERARE LO STATO*)
tempConfrontoAlive:= Sys.Time_CT_DT - LastSeen;
tempConfronto:=                 (desideredState.ID_Geolumen=feedbackState.ID_Geolumen) AND
					  (desideredState.DimmValue_0=feedbackState.DimmValue_0) AND
 					  (desideredState.DimmValue_1=feedbackState.DimmValue_1) AND
					  (desideredState.DimmValue_2=feedbackState.DimmValue_2) ;
IF NOT (USING_EXTERNAL_ASTRO AND desideredState.DimmValue_0 = 0) THEN
	IF( (tempConfrontoAlive>=TIME_NO_FEEBACK_RESEND_STATUS OR tempConfronto=FALSE) AND (retryStatusNotAligned<MAX_RETRY_STATUS_NOT_ALIGNED AND IS_PRE_GLOBAL_ON_ONGOING=FALSE)) THEN
		doAlignStatus();
	ELSIF (tempConfrontoAlive<TIME_NO_FEEBACK_RESEND_STATUS AND tempConfronto=TRUE AND IS_PRE_GLOBAL_ON_ONGOING=FALSE) THEN
		retryStatusNotAligned:=0;
	END_IF
END_IF

(*GESTIONE LOG EV PER NODO STATO DISALLINEATO/RIALLINEATO *)
fltNodeStatusNotAligned(IN:=(isGeolumenEqualStatus(desideredState,feedbackState)=FALSE)  AND retryStatusNotAligned>=MAX_RETRY_STATUS_NOT_ALIGNED);
IF fltNodeStatusNotAligned.EVH THEN
	LogEv(EL_Alarm,EO_LUX,ID_Lux,14,'Geolumen node with desidered status DIFFERENT from feedback status');
END_IF
IF fltNodeStatusNotAligned.EVL THEN
	LogEv(EL_Log,EO_LUX,ID_Lux,15,'Geolumen node with desidered status = feedback status');
	retryStatusNotAligned:=0;
END_IF
END_ACTION
ACTION doAlignStatus:
(*invia periodicamente re-set in caso di stato non allineato *)
timerAlignStatus(IN:=NOT timerAlignStatus.Q,PT:=TIME_WAIT_RETRY_NOT_ALIGNED);
IF isCoordinatorBooted() AND timerAlignStatus.Q THEN

	IF NOT DEBUG_NO_CONTROL_LIGHTS THEN

		SendDataQueue(pTxData:=ADR(toSendSetString));
		SendDataQueue.addMessage();
		(*SendDataQueue(pTxData:=ADR(toSendGetString)); (* <=== GET SUCCESSIVA EVITATA *)
		SendDataQueue.addMessage();*)

	END_IF

	retryStatusNotAligned:=retryStatusNotAligned+1;
END_IF
END_ACTION
ACTION resetLampIndicators:
GlobalMaxCurrent	:=0;
GlobalMaxVoltage:=0;
GlobalMaxPower:=0;
dayFeed:=0;
END_ACTION
ACTION resetRetryCounters:
(*reset di tutti i contatori di tentativi fatti *)
retryDisappear:=0;
retryStatusNotAligned:=0;
END_ACTION
ACTION updateDesideredState:
(*calcolo stato desiderato a partire dal desideredDimmValue*)
desideredState.id_Geolumen:=ID_Geolumen;
(*normalizzo: dal valore desiderato 0-100 alla scala effettova del nodo geolumen*)
normalizedDesideredDimmValueGeoLumen:=(WORD_TO_REAL(desideredDimmValue)/WORD_TO_REAL(MAX_DIMM_LUX_CLEVERGY))*MAX_DIMM;
(*lo applico a tutti i canali PWM*)
desideredState.DimmValue_0:=REAL_TO_WORD(normalizedDesideredDimmValueGeoLumen);
desideredState.DimmValue_1:=REAL_TO_WORD(normalizedDesideredDimmValueGeoLumen);
desideredState.DimmValue_2:=REAL_TO_WORD(normalizedDesideredDimmValueGeoLumen);

(*definisco la stringa di set e get per il nodo corrente V1*)(*old*)
IF GEOLUMEN_COORD_VERSION =1 THEN

	templateDimm:=',x,x,x$R';
	tmpNum:=WORD_TO_STRING(REAL_TO_WORD(normalizedDesideredDimmValueGeoLumen));
	commandString:=REPLACE_ALL(templateDimm,'x',tmpNum);
	sendString := 'NDE_SET_LIGHT=';
	sendString:=CONCAT(SendString, DWORD_TO_STRING(ID_Geolumen));
	sendString:=CONCAT(SendString, commandString);
	toSendSetString:=sendString;
	templateGet:='NDE_GET_STATUS=x$R';
	toSendGetString:=REPLACE_ALL(templateGet,'x',DWORD_TO_STRING(ID_Geolumen));

ELSIF GEOLUMEN_COORD_VERSION =2 THEN

	templateDimm:='=x,x,x$R';
	tmpNum:=WORD_TO_STRING(REAL_TO_WORD(normalizedDesideredDimmValueGeoLumen));
	commandString:=REPLACE_ALL(templateDimm,'x',tmpNum);
	sendString := 'NDE_SET_LIGHT:';
	sendString:=CONCAT(SendString, DWORD_TO_STRING(ID_Geolumen));
	sendString:=CONCAT(SendString, commandString);
	toSendSetString:=sendString;
	templateGet:='NDE_GET_STATUS:x$R';
	toSendGetString:=REPLACE_ALL(templateGet,'x',DWORD_TO_STRING(ID_Geolumen));

END_IF
END_ACTION
ACTION updateEchoState:
echoLastSeen:=Sys.Time_CT_DT;
END_ACTION
ACTION updateFeedbackState:
(*aggiorno lo stato interno del nodo e del LUX correlato *)
dayFeed:=dayFeed+1;
lastSeen:=Sys.Time_CT_DT;
lastPar:=feedbackState.lastPar;
(*resetto il contatore di nodo alive*)
retryDisappear:=0;
(*determino il valore rilevato dal campo - considero solo il canale pwm 0*)
fTemp1:=WORD_TO_REAL(feedbackState.DimmValue_0);
fTemp2:=WORD_TO_REAL(MAX_DIMM);
fTemp3:=WORD_TO_REAL(MAX_DIMM_LUX_CLEVERGY);
fTemp4:=(fTemp1/fTemp2)*fTemp3;
fNormValue:=REAL_TO_WORD(fTemp4);


IF(feedbackState.lampPower>GlobalMaxPower) THEN GlobalMaxPower:=feedbackState.lampPower; END_IF
IF(feedbackState.lampCurrent>GlobalMaxCurrent) THEN GlobalMaxCurrent:=feedbackState.lampCurrent; END_IF
IF(feedbackState.lampVoltage>GlobalMaxVoltage) THEN GlobalMaxVoltage:=feedbackState.lampVoltage; END_IF

lampBroken:=dayFeed>2 AND (GlobalMaxPower<5 AND  GlobalMaxCurrent<30);

(*aggiorno lo stato del LUX relativo al nodo corrente*)
FOR i:=1 TO MAX_LUXNUM DO

	IF LuxElement[i].ID <> 0 AND LuxElement[i].ID=ID_Lux THEN

		LuxElement[i](Lux_State:=(fNormValue>0),
					Lux_StateAnalog:=fNormValue,
					WorkingTime:=GlobalWorkingtime[i],
					PowerOnCycles:=GlobalPowerOnCycles[i],
					EnergyCounter:=GlobalEnergyCounter[i],
					EnergyCounter_t:=GlobalEnergyCounter_t[i],KeyQty:=2);

	END_IF

END_FOR
END_ACTION

(* POU obj_LUX/obj_LUX, ST *)
FUNCTION_BLOCK obj_LUX
(*
   v1.0[feb-2016] - Create GIURE      
	
   Info:
   	
*)
VAR CONSTANT
	(*Costant in lux obj*)
	NO_DIMMING	: BYTE:=0;
	DIMMING		: BYTE:=1;
	ROT			: BOOL:=1;
	GRUN		: BOOL:=0;
	MAX_DIMM_VALUE:WORD:=100;
END_VAR

VAR_INPUT
	Status_Log		: INT;
	(* Settings *)
	ID					: DWORD;
	DimmingType		: BYTE;	 (* 0: no dimming (digital), 1: dimming (analog) *)
	DimmingValForTimer	: INT;	 (* valore 0...100 del dimming di default del lux sotto timer *)
	DimmingValForManual    : INT;           (*valore 0...100 del dimming di default del lux in manuale *)
	(* Controls *)
	CTRL_MODE			: en_Modality;	 (* 0:MAN OFF, 1:MAN-ON, 3:Timer laser, 2:Cronografo*)
	CTRL_MODE_BackUp	: en_Modality;	 (*Salvo il valore di default per il ripristino *)
	LuxTimer		: TIME; (* Tempo di accensione del lux settato nella tabella TabLuxPsg ottenuta dal file di config su SD *)
	HourMinStartOn	: TOD; (* Orario di start per rilevazione sensori start timer (Mode 03) *)
	HourMinEndOn	: TOD; (* Orario di end per rilevazione sensori start timer (Mode 03) *)
	ValInCronoInLux : INT;	(* Valore del setpoint arrivato dal crono *)
	RefTableAutLuxPsg : WORD; (* indice di riferimento alla tabella AUT_LUX_PSG se mode = 3 *)
	RestoreKey		: BOOL; (* se attivato viene ripristinato il mode di default *)
	CtrlTrig		: BOOL; (* Trigger for timer start *)
	CtrlKeyList		: ARRAY [0..9] OF BOOL; (* External KEY control input *)
	CtrlExton : BOOL ;
	KeyQty			: BYTE; (* numero di key all'ingresso *)
	KeyMode			: en_KeyMode;	(* BYTE; //Modalità di funzionamento richiesta dal key *)
	DimmingValForKeyList: ARRAY [0..9] OF INT;
	DimmingValForKeyMax: BOOL; (* Se TRUE --> si sceglie il valore massimo; Se FALSE --> si sceglie il valore minimo *)
	ActionKey		: en_ActionKey; (* 00-NormalMode, 01-SwitchON, 02-SwitchOFF, 03-Restore *)
	(* Physical inputs *)
	Lux_State		: BOOL; 	          (* Status on/off feedback *)
	Lux_StateAnalog	: WORD;   (* Status dimming feedback *)

END_VAR
VAR_IN_OUT
	WORKINGTIME		: DWORD; (* [sec] Internal working time counter *)
	POWERONCYCLES		: WORD;	(* DWORD; Internal counter of power-on cycles *)
	ENERGYCOUNTER		: WORD;	(* DWORD;  [E-1 kWh] Internal energy counter *)
	ENERGYCOUNTER_t 	: DWORD; (* Temporary energy in E-2*Wsec *)
END_VAR
VAR_OUTPUT
	(* Physical outputs *)
	LuxDigitalOut	: BOOL;
	LuxAnalogOut	: WORD;
	LuxTypeOut		: BOOL;
	Lux_Enable		: BOOL;	(*  uscita logica per compatibilità con sw preesistente (ex (* Control output *)) *)
	Lux_EnableAnalog : WORD;      (*  uscita enable dimming *)
	(* Status *)
	Status_Vis 		: DWORD;
END_VAR
VAR
	TickTimer		: TON := ( PT:=T#1S );
	TrigTimer		: TOF ;

	KeyTimer		: TIME := T#200ms;
	sLux_EN			: FLT_EVENT;
	chkLux_ST			: FLT_TIME := ( TTAP:=T#20S, INITEV:=FALSE );
	chkLux_ST_Analog		: FLT_TIME := ( TTAP:=T#20S, INITEV:=FALSE );
	HourMinNow		: STRING;
	semaphore		: BOOL:=GRUN;
	OnFromKey		: BOOL;
	fTrigFun		: F_TRIG;
	rTrigFun		: R_TRIG;
	fTrigKey		: F_TRIG;
	ActionKeyState	: en_ActionKey;
	KeyCounter, x	: BYTE;
	CtrlKey			: BOOL;
	DimmingValForKey: INT; (* valore 0...100 del dimming di default del lux sotto key *)
	ModeToServer : BYTE;
	ForcedOn : BYTE;
	ForcedOff : BYTE;
END_VAR
VAR CONSTANT

	COLOR_RED			: DWORD	:= 16#2020F0;
	COLOR_YELLOW		: DWORD	:= 16#20F0F0;
	COLOR_GREEN			: DWORD	:= 16#20F020;
	COLOR_GREEN_OFF		: DWORD := 16#006000;
END_VAR
(* Con l'ID si identifica il numero del lux sul campo quindi il suo valore può variare da 1 a LUXM_MAX (attualmente 1...900) *)
IF (KeyMode = BUTTON_NO) OR (KeyMode = BUTTON_NC) THEN (* se si usano dei pulsanti sui vari digital input...*)
	KeyCounter := 0;
	FOR x:=0 TO  KeyQty-1 DO
		IF CtrlKeyList[x] = 1 THEN
			KeyCounter := KeyCounter + 1;
		END_IF
	END_FOR
	IF (KeyCounter MOD 2) = 0 THEN
		CtrlKey := FALSE;
	ELSE
		DimmingValForKey := DimmingValForKeyList[0]; (* In caso di pulsanti si prende il valore della posizione 0 dell'array *)
		CtrlKey := TRUE;
	END_IF
ELSE (* altrimenti se uso l'interruttore ne posso usare solo 1 nella posizione 0 dell'array *)
	IF (DimmingValForKeyMax) THEN
		DimmingValForKey := 0;
		FOR x:=0 TO  KeyQty-1 DO
			IF (CtrlKeyList[x] = 1) AND (DimmingValForKeyList[x] > DimmingValForKey)
			THEN
				DimmingValForKey := DimmingValForKeyList[x];
			END_IF
		END_FOR
	ELSIF NOT(DimmingValForKeyMax) THEN
		DimmingValForKey :=MAX_DIMM_VALUE;
		FOR x:=0 TO  KeyQty-1 DO
			IF (CtrlKeyList[x] = 1) AND (DimmingValForKeyList[x] < DimmingValForKey)
			THEN
				DimmingValForKey := DimmingValForKeyList[x];
			END_IF
		END_FOR
	END_IF
	CtrlKey := 0;
	FOR x:=0 TO  KeyQty-1 DO
			CtrlKey := CtrlKey OR CtrlKeyList[x];
	END_FOR

END_IF

CASE DimmingType OF (* set dell' AsiTypeOut per sapere se eseguire il set di un analog out o di un digital out *)
	NO_DIMMING:	(* if no dimming we are using a digital output *)
		LuxTypeOut := DIGITAL; (* Set digital out mode *)
	DIMMING:	(*  if dimming we are using analog output *)
		LuxTypeOut := ANALOG; (* Set analog out mode *)
END_CASE

(* Control logic *)
(* Restore mode and value	*)
IF RestoreKey THEN
	CTRL_MODE := CTRL_MODE_BackUp;
END_IF

CASE CTRL_MODE OF
	ManualeOff: (*  0 Manuale Off *)
		(* Se commutazione arrivata da key durante funzionamento in timer o cronografo *)
		IF  NOT(CtrlKey) AND (ActionKey > NormalMode) AND ( ActionKeyState = SwitchOFF)THEN
			ActionKeyState := NormalMode;
			CTRL_MODE := CTRL_MODE_BackUp;
		ELSE
			CASE DimmingType OF
				NO_DIMMING:	(* if no dimming we are using a digital output *)
					LuxDigitalOut := TRUE; (* Lux spento (digital) *)
				DIMMING:	(*  if dimming we are using analog and digital output *)
					DimmerCtrl(); (* In caso di switch off in manuale è sempre zero anche se arriva da key *)
			END_CASE
		END_IF
	ManualeOn: (*  1 Manuale On *)
		(* Se commutazione arrivata da key durante funzionamento in timer o cronografo *)
		IF  NOT(CtrlKey) AND (ActionKey > NormalMode) AND ( ActionKeyState = SwitchON) THEN
			ActionKeyState := NormalMode;
			CTRL_MODE := CTRL_MODE_BackUp;
		ELSE
			CASE DimmingType OF
				NO_DIMMING:	(* if no dimming we are using a digital output *)
					LuxDigitalOut := FALSE; (* Lux acceso (digital) *)
				DIMMING:	(*  if dimming we are using analog and digital output  *)
					IF ActionKeyState = SwitchON THEN
						DimmerCtrlKeyOn(); (* Se il manuale on è settato a causa di un key si impongono i dati del key stesso *)
					ELSE
						DimmerCtrl();
					END_IF
			END_CASE
		END_IF
	Cronografo: (*  2 Cronografo *)
		IF  (CtrlKey) AND (ActionKey > NormalMode) THEN
			CASE  ActionKey OF
				SwitchON: 	(* Corrisponde al manuale ON *)
					CTRL_MODE := ManualeOn;
					ActionKeyState := SwitchON;
					CASE DimmingType OF
						NO_DIMMING:	(* if no dimming we are using a digital output *)
							LuxDigitalOut := FALSE; (* Lux acceso (digital) *)
						DIMMING:	(*  if dimming we are using analog and digital output  *)
							DimmerCtrlKeyOn();
					END_CASE

				SwitchOFF:	(* Corrisponde al manuale OFF  *)
					CTRL_MODE := ManualeOff;
					ActionKeyState := SwitchOFF;
					CASE DimmingType OF
						NO_DIMMING:	(* if no dimming we are using a digital output  *)
							LuxDigitalOut := TRUE; (* Lux spento (digital)  *)
						DIMMING:	(*  if dimming we are using analog and digital output  *)
							DimmerCtrlKeyOff();
					END_CASE
			END_CASE
		ELSE
			CASE DimmingType OF
				NO_DIMMING:	(* if no dimming we are using a digital output  *)
					IF ValInCronoInLux = MAX_DIMM_VALUE (* OR ( LuxElement[i].PressKeyVisuOn)  *)
						THEN
						LuxDigitalOut := FALSE; (* Lux acceso (digital)  *)
						ELSE IF ValInCronoInLux = 0 (* OR ( NOT LuxElement[i].PressKeyVisuOn)  *)
							THEN
							LuxDigitalOut := TRUE; (* Lux spento (digital)  *)
						END_IF
					END_IF
				DIMMING:	(*  if dimming we are using analog output  *)
					DimmerCtrl();
			END_CASE
		END_IF
	Timer: (*  3 Timer   *)
	IF  (CtrlKey) AND (ActionKey > NormalMode) THEN
		CASE  ActionKey OF
			SwitchON: 	(* Corrisponde al manuale ON  *)
				CTRL_MODE := ManualeOn;
				ActionKeyState := SwitchON;
				CASE DimmingType OF
					NO_DIMMING:	(* if no dimming we are using a digital output  *)
						LuxDigitalOut := FALSE; (* Lux acceso (digital)  *)
					DIMMING:	(*  if dimming we are using analog and digital output   *)
						DimmerCtrlKeyOn();
				END_CASE

			SwitchOFF:	(* Corrisponde al manuale OFF  *)
				CTRL_MODE := ManualeOff;
				ActionKeyState := SwitchOFF;
				CASE DimmingType OF
					NO_DIMMING:	(* if no dimming we are using a digital output  *)
						LuxDigitalOut := TRUE; (* Lux spento (digital)  *)
					DIMMING:	(*  if dimming we are using analog and digital output  *)
						DimmerCtrlKeyOff();
				END_CASE
		END_CASE
	ELSE
		CASE DimmingType OF
			NO_DIMMING:	(* if no dimming we are using a digital output  *)
				HourMinNow:=CONCAT('TOD#', BYTE_TO_STRING(Sys.Time_Hour));
				HourMinNow:=CONCAT(HourMinNow, ':');
				HourMinNow:=CONCAT(HourMinNow, BYTE_TO_STRING(Sys.Time_Min));
				HourMinNow:=CONCAT(HourMinNow,':00');

				(* Trig timer *)
				TrigTimer.PT:=LuxTimer;
				TrigTimer(IN:= CtrlTrig);

				IF (((STRING_TO_TOD(HourMinNow) > HourMinStartOn) AND (STRING_TO_TOD(HourMinNow) < HourMinEndOn))  (* Se siamo nell'orario corretto  *)
				OR ((LuxDigitalOut = FALSE) AND (TrigTimer.Q = FALSE))) (* oppure si era acceso e adesso siamo passati fuori orario e dobbiamo spegnere  *)
				THEN
					IF TrigTimer.Q THEN
						LuxDigitalOut := FALSE; (* Lux acceso (digital)  *)
						ELSE
							LuxDigitalOut:= TRUE; (* Lux spento (digital)  *)
					END_IF
				END_IF
			DIMMING:	(*  if dimming we are using analog output  *)

				HourMinNow:=CONCAT('TOD#', BYTE_TO_STRING(Sys.Time_Hour));
				HourMinNow:=CONCAT(HourMinNow, ':');
				HourMinNow:=CONCAT(HourMinNow, BYTE_TO_STRING(Sys.Time_Min));
				HourMinNow:=CONCAT(HourMinNow,':00');

				(* Trig timer *)
				TrigTimer.PT:=LuxTimer;
				TrigTimer(IN:= CtrlTrig);

				IF (((STRING_TO_TOD(HourMinNow) > HourMinStartOn) AND (STRING_TO_TOD(HourMinNow) < HourMinEndOn))  (* Se siamo nell'orario corretto  *)
				OR ((LuxDigitalOut = FALSE) AND (TrigTimer.Q = FALSE))) (* oppure si era acceso e adesso siamo passati fuori orario e dobbiamo spegnere  *)
				THEN
					IF TrigTimer.Q THEN
						DimmerCtrl(); (* Lux acceso  *)
						ELSE
							LuxAnalogOut := 0; (* Lux spento  *)
							LuxDigitalOut := TRUE; (* Lux spento (digital)  *)
					END_IF
				END_IF
		END_CASE
		END_IF
	KeyControl: (*  4 Key function  *)
		IF CtrlKey THEN
			CASE DimmingType OF
				NO_DIMMING:	(* if no dimming we are using a digital output  *)
					LuxDigitalOut := FALSE; (* Lux acceso (digital)  *)
				DIMMING:	(*  if dimming we are using analog and digital output   *)
					DimmerCtrlKeyOn();
			END_CASE
		ELSIF CtrlKey = 0 THEN
			CASE DimmingType OF
				NO_DIMMING:	(* if no dimming we are using a digital output  *)
					LuxDigitalOut := TRUE; (* Lux spento (digital)  *)
				DIMMING:	(*  if dimming we are using analog and digital output  *)
					DimmerCtrlKeyOff();
			END_CASE
		END_IF
	END_CASE

(* ----------------------------------------------------------------------------------------------------------------------------------------  *)
(* Se i pin del feedback relè non sono cavallottati si usa la seguente riga al posto di quelle successive indicate da(#)  *)
(* REL_ST := LUX_ST[ID];	  																					 *)
(* ----------------------------------------------------------------------------------------------------------------------------------------   *)

(* setting della variabile REL_EN per compatibilità con il sw preesistente  *)
CASE DimmingType OF
	NO_DIMMING:	(* if no dimming we are using a digital output  *)
	IF LuxDigitalOut = TRUE  (* Lux spento  *)
		THEN
			(* Lux_State := FALSE;	//A causa del cavallotto sui pin del relè forzo a falso (#)  *)
			(* Lux_State := LUX_ST[ID];	  *)
			Lux_Enable := FALSE;
		ELSIF LuxDigitalOut = FALSE  (* Lux acceso			   *)
			THEN
				(* Lux_State := LUX_ST[ID];	//Quando so che la luce è accesa leggo lo stato del pin (che essendo cavallottato sarà a 1) (#)  *)
				Lux_Enable := TRUE;
	END_IF

	DIMMING:	(*  if dimming we are using analog output  *)
	IF LuxAnalogOut  = 0 (* Lux spento				  *)
		THEN
			(* REL_ST := FALSE;	 A causa del cavallotto sui pin del relè forzo a falso (#)  *)
			(* Lux_State := LUX_ST[ID];	  *)
			Lux_Enable := FALSE;
			Lux_EnableAnalog := LuxAnalogOut; (*GIURE ver 008*)
		ELSIF LuxAnalogOut > 0  (* Lux acceso			  *)
			THEN
				(* Lux_State := LUX_ST[ID];	 Quando so che la luce è accesa leggo lo stato del pin (che essendo cavallottato sarà a 1) (#)  *)
				Lux_Enable := TRUE;
				Lux_EnableAnalog := LuxAnalogOut; (*GIURE ver 008*)
	END_IF

END_CASE
(* Temporary energy counter *)
TickTimer(IN:=NOT TickTimer.Q);
IF TickTimer.Q AND Lux_Enable THEN
	WORKINGTIME:=WORKINGTIME+1;
	IF ENERGYCOUNTER_t>36000000 THEN
		ENERGYCOUNTER_t:=ENERGYCOUNTER_t-36000000;
		ENERGYCOUNTER:=ENERGYCOUNTER+1;
	END_IF
END_IF

(* Generate status events *)
sLux_EN(IN:=Lux_Enable);
IF sLux_EN.EVL THEN
	LogEv(EL_Log,EO_LUX,ID,2,'Light OFF'); (* Light OFF  *);
END_IF
IF sLux_EN.EVH THEN
	LogEv(EL_Log,EO_LUX,ID,3,'Light ON'); (* Light ON  *);
	POWERONCYCLES:=POWERONCYCLES+1;
END_IF

(* Check status feedback *)
chkLux_ST_Analog(IN:=(Lux_StateAnalog<>Lux_EnableAnalog));
IF chkLux_ST_Analog.EVH THEN
	LogEv(EL_Alarm,EO_LUX,ID,9,CONCAT(CONCAT(CONCAT('Fail Analog, exp:',WORD_TO_STRING(Lux_EnableAnalog)),' found'),WORD_TO_STRING(Lux_StateAnalog))); (* Feedback failure - Lux_StateAnalog<>Lux_EnableAnalog *)
END_IF

IF chkLux_ST_Analog.EVL THEN
	LogEv(EL_Log,EO_LUX,ID,1,'Successful Analog'); (* Light feedback OK - Lux_StateAnalog = Lux_EnableAnalog *)
END_IF


(* Check status feedback *)
chkLux_ST(IN:=(Lux_State<>Lux_Enable));
IF chkLux_ST.EVH THEN
	LogEv(EL_Alarm,EO_LUX,ID,9,'Fail'); (*  Feedback failure - Lux_State<>Lux_Enable  *);
END_IF
IF chkLux_ST.EVL THEN
	LogEv(EL_Log,EO_LUX,ID,1,'Successful'); (*  Light feedback OK - Lux_State = Lux_Enable  *);
END_IF


(* Status color *)
IF Status_Log=1 THEN
	Status_Vis:=COLOR_YELLOW;
ELSIF Status_Log=2 THEN
	Status_Vis:=COLOR_RED;
ELSE
	Status_Vis:=SEL(Lux_Enable,COLOR_GREEN_OFF,COLOR_GREEN);
END_IF
END_FUNCTION_BLOCK
ACTION AddLogData:
Logger.s1:=INSERT('&LUX=',DWORD_TO_STRING(ID),4);
IF ID<10 THEN Logger.s1:=INSERT(Logger.s1,'0',4); END_IF

(*Logger.s1:=CONCAT(Logger.s1,WORD_TO_STRING(REL_V));				Logger.s1:=CONCAT(Logger.s1,';');
//Logger.s1:=CONCAT(Logger.s1,WORD_TO_STRING(REL_A));				Logger.s1:=CONCAT(Logger.s1,';');
//Logger.s1:=CONCAT(Logger.s1,DWORD_TO_STRING(ENERGYCOUNTER));	Logger.s1:=CONCAT(Logger.s1,';');*)

Logger.s1:=CONCAT(Logger.s1,BOOL_TO_STRING(Lux_Enable));			Logger.s1:=CONCAT(Logger.s1,';');
Logger.s1:=CONCAT(Logger.s1,DWORD_TO_STRING(WorkingTime));		Logger.s1:=CONCAT(Logger.s1,';');
Logger.s1:=CONCAT(Logger.s1,DWORD_TO_STRING(PowerOnCycles));	Logger.s1:=CONCAT(Logger.s1,';');
(*//Logger.s1:=CONCAT(Logger.s1,INT_TO_STRING(REL_TEMP));			Logger.s1:=CONCAT(Logger.s1,';');*)

CASE CTRL_MODE OF
	0: 	(* Manuale OFF *)
		ModeToServer := 0;
		ForcedOn := 0;
		ForcedOff := 1;
	1:	(* Manuale ON *)
		ModeToServer := 0;
		ForcedOn := 1;
		ForcedOff := 0;	
	2:	(* Cronografo *)
		ModeToServer := 2;
		ForcedOn := 0;
		ForcedOff := 0;
	3: 	(* Timer *)
		ModeToServer := 3;
		ForcedOn := 0;
		ForcedOff := 0;
END_CASE

Logger.s1:=CONCAT(Logger.s1,BYTE_TO_STRING(ModeToServer));			Logger.s1:=CONCAT(Logger.s1,';');
Logger.s1:=CONCAT(Logger.s1,INT_TO_STRING(Status_Log));			Logger.s1:=CONCAT(Logger.s1,';');
Logger.s1:=CONCAT(Logger.s1,BYTE_TO_STRING(ForcedOn));			Logger.s1:=CONCAT(Logger.s1,';');
Logger.s1:=CONCAT(Logger.s1,BYTE_TO_STRING(ForcedOff));			Logger.s1:=CONCAT(Logger.s1,';');
Logger.s1:=CONCAT(Logger.s1,BYTE_TO_STRING(DimmingType));		Logger.s1:=CONCAT(Logger.s1,';');
Logger.s1:=CONCAT(Logger.s1,WORD_TO_STRING(Lux_EnableAnalog));

ADDSTRING(ADR(Logger.TData), ADR(Logger.s1), Logger.TLen);
END_ACTION
ACTION DimmerCtrl:
CASE CTRL_MODE OF
	0: (* Manuale Off *)
		LuxAnalogOut := 0; (* Lux spento *)
		LuxDigitalOut := TRUE; (* Lux spento (digital) *)

	1: (* Manuale On *)
       		(* IF DimmingValForManual > 0 THEN    (*modifica ver 007 per dimmer su comando manuale on *)
           		 LuxDigitalOut := FALSE;  (*Lux acceso (digital)*)
       		 END_IF*)

		IF  DimmingValForManual>MAX_DIMM_VALUE THEN
			LuxAnalogOut := MAX_DIMM_VALUE;
        		ELSE
			LuxAnalogOut := INT_TO_WORD(DimmingValForManual);  (* Lux acceso *)
		END_IF

		LuxDigitalOut := FALSE; (* Lux acceso (digital) *)
	2: (* Cronografo *)
		IF ValInCronoInLux > 0 THEN
			LuxDigitalOut := FALSE; (* Lux acceso (digital) *)
		ELSE
			LuxDigitalOut := TRUE; (* Lux spento (digital) *)
		END_IF
		IF (ValInCronoInLux>MAX_DIMM_VALUE) THEN (* al massimo MAX_DIMM_VALUE*)
			LuxAnalogOut:=MAX_DIMM_VALUE;
		ELSE
			LuxAnalogOut := INT_TO_WORD(ValInCronoInLux);
		END_IF
	3: (* Timer 		 *)
		IF DimmingValForTimer > 0 THEN
			LuxDigitalOut := FALSE; (* Lux acceso (digital) *)
		ELSE
			LuxDigitalOut := TRUE; (* Lux spento (digital) *)
		END_IF
		IF (DimmingValForTimer>MAX_DIMM_VALUE) THEN
			LuxAnalogOut := MAX_DIMM_VALUE;
		ELSE
			LuxAnalogOut := INT_TO_WORD(DimmingValForTimeR);
		END_IF

	ELSE (* default *)
		LuxDigitalOut := FALSE; (* Lux acceso (digital) *)
		LuxAnalogOut := MAX_DIMM_VALUE;
END_CASE
END_ACTION
ACTION DimmerCtrlKeyOff:
LuxAnalogOut := 0; (*Lux spento*)
LuxDigitalOut := TRUE; (*Lux spento (digital)*)
END_ACTION
ACTION DimmerCtrlKeyOn:
IF (INT_TO_WORD(DimmingValForKey)>MAX_DIMM_VALUE) THEN
	LuxAnalogOut := MAX_DIMM_VALUE;
ELSE
	LuxAnalogOut := INT_TO_WORD(DimmingValForKey);
END_IF
LuxDigitalOut := FALSE; (*Lux acceso (digital) *)
END_ACTION
ACTION StatReset:
(* Reset statistic counters *)
WORKINGTIME:=0;
POWERONCYCLES:=0;
ENERGYCOUNTER:=0;
END_ACTION

(* POU PLANTCONFIG/objAstroLog, ST *)
(* logga una sequenza di ASTR identifica da una riga *)
FUNCTION objAstroLog:BOOL
VAR CONSTANT
	GROUP_SIZE: INT:=10; (*FACTOR OF GROUPING*)
END_VAR
VAR_INPUT
	(*numero riga *)
	partenza:WORD;
END_VAR
VAR
	(*elementi per riga *)

	groupNumber : WORD;
	i : WORD;
	j : WORD;
	index:WORD;
	isObj : BOOL;
	lastGroup:WORD:=0;
END_VAR
i:=partenza-1;

(*verifico se nel gruppo corrente c'è qualche ASTR valido *)
isObj:=FALSE;
FOR j:=1 TO GROUP_SIZE DO
	index:=i*GROUP_SIZE+j;
	IF(index>0 AND index<=MAX_LUXNUM AND ASTR[index].ID<>0 ) THEN isObj:=TRUE; j:=GROUP_SIZE; END_IF
END_FOR

(* se c'è qualche ASTR valido da fare, procedo *)
IF(isObj) THEN
	Logger_Head();
	FOR j:=1 TO GROUP_SIZE DO
		index:=i*GROUP_SIZE+j;
		IF(index>0 AND index<=MAX_LUXNUM AND ASTR[index].ID<>0 ) THEN ASTR[index].AddLogData(); END_IF
	END_FOR
	Logger_Send();
END_IF
END_FUNCTION

(* POU PLANTCONFIG/objLuxLog, ST *)
(* logga una sequenza di LUX identifica da una riga *)
FUNCTION objLuxLog:BOOL
VAR CONSTANT
	GROUP_SIZE: INT:=10; (*FACTOR OF GROUPING*)
END_VAR
VAR_INPUT
	partenza:WORD;
END_VAR
VAR
	groupSize: WORD:=10; (*FACTOR OF GROUPING*)
	groupNumber : WORD;
	i : WORD;
	j : WORD;
	index:WORD;
	isObj : BOOL;
	lastGroup:WORD:=0;
END_VAR
i:=partenza-1;

(*verifico se nel gruppo corrente c'è qualche LUX valido *)
isObj:=FALSE;
FOR j:=1 TO GROUP_SIZE DO
	index:=i*GROUP_SIZE+j;
	IF(index>0 AND index<=MAX_LUXNUM AND LuxElement[index].ID<>0 ) THEN isObj:=TRUE; j:=GROUP_SIZE; END_IF
END_FOR

(* se c'è qualche LUX valido da fare, procedo *)
IF(isObj) THEN
	Logger_Head();
	FOR j:=1 TO GROUP_SIZE DO
		index:=i*GROUP_SIZE+j;
		IF(index>0 AND index<=MAX_LUXNUM AND LuxElement[index].ID<>0 ) THEN

			LuxElement[index].AddLogData(WORKINGTIME:=GlobalWorkingtime	[index],
									    POWERONCYCLES:=GlobalPowerOnCycles[index],
									    ENERGYCOUNTER:=GlobalEnergyCounter[index],
									    ENERGYCOUNTER_t :=GlobalEnergyCounter_t[index]);

		END_IF
	END_FOR
	Logger_Send();
END_IF
END_FUNCTION

(* POU ClevergyUtils/Utils Functions/PLANT_STATUS, ST *)
FUNCTION_BLOCK PLANT_STATUS
VAR_INPUT
	obj_Status		:	WORD;
END_VAR
VAR_OUTPUT
	plantStatus		:	WORD;
END_VAR
VAR
	Pwm				:	TON := (PT:=T#1s);
END_VAR
(*CASE plantStatus OF

	0:	(* Plant OK - Everything works well *)
		Pwm(IN:=FALSE);							(* Stop timer if running *)
		LAMP_AL := FALSE;						(* Keep the lamp switched off *)

	1:	(* Plant in warning *)
		Pwm(IN:= NOT(Pwm.Q));

		IF Pwm.Q THEN
			LAMP_AL := NOT LAMP_AL;				(* Toggle output *)
		END_IF

	2:	(* Plant in alarm *)
		Pwm(IN:=FALSE);							(* Stop timer if running *)
		LAMP_AL	:= TRUE;						(* Keep the lamp switched on *)

END_CASE*)

plantStatus := 0;		(* Reset plant status *)
END_FUNCTION_BLOCK
ACTION UpdateStatus:
IF plantStatus = 2 THEN

	RETURN;					(* If plant already in alarm condition do nothing *)

ELSE
	IF obj_Status <> 0 THEN
		plantStatus := obj_Status;			(* If plant in warning/normal condition and current object in alarm, update plant status *)
	END_IF
END_IF
END_ACTION

(* POU ClevergyUtils/PLC_WDT, ST *)
FUNCTION PLC_WDT: DWORD VAR_INPUT dwEvent: DWORD; dwFilter: DWORD; dwOwner: DWORD; END_VAR
LogEv(EL_AlarmStop,EO_SYS,1,10,'Watchdog');
END_FUNCTION

(* POU ClevergyUtils/Utils Functions/RAW16TOHEXSTR, ST *)
FUNCTION RAW16TOHEXSTR : STRING(128)
VAR_INPUT
	pData: POINTER TO BYTE;
	DataLen: BYTE;
END_VAR
VAR
	pt: POINTER TO BYTE;
	xl: BYTE;
END_VAR
pt:=ADR(RAW16TOHEXSTR);
xl:=0;

WHILE DataLen>0 AND xl<120 DO

	pData:=pData+1;

	pt^ := (pData^ / 16#10) + 48 + (((pData^ / 16#10)/10)*7);
	pt:=pt+1;
	pt^ := (pData^ AND 16#0F)  + 48 + (((pData^ AND 16#0F)/10)*7);
	pt:=pt+1;

	pData:=pData-1;

	pt^ := (pData^ / 16#10) + 48 + (((pData^ / 16#10)/10)*7);
	pt:=pt+1;
	pt^ := (pData^ AND 16#0F)  + 48 + (((pData^ AND 16#0F)/10)*7);
	pt:=pt+1;

	xl:=xl+4;

	DataLen:=DataLen-2;
	pData:=pData+2;

END_WHILE

pt^:=0;
END_FUNCTION

(* POU ClevergyUtils/RAWTOHEXSTR, ST *)
FUNCTION RAWTOHEXSTR : STRING(128)
VAR_INPUT
	pData: POINTER TO BYTE;
	DataLen: BYTE;
END_VAR
VAR
	pt: POINTER TO BYTE;
	xl: BYTE;
END_VAR
pt:=ADR(RAWTOHEXSTR);

xl:=2;

WHILE DataLen>0 AND xl<128 DO

	pt^ := (pData^ / 16#10) + 48 + (((pData^ / 16#10)/10)*7);
	pt:=pt+1;
	pt^ := (pData^ AND 16#0F)  + 48 + (((pData^ AND 16#0F)/10)*7);
	pt:=pt+1;

	xl:=xl+2;

	DataLen:=DataLen-1;
	pData:=pData+1;

END_WHILE

pt^:=0;
END_FUNCTION

(* POU ClevergyUtils/RESET_ARRAY, ST *)
FUNCTION RESET_ARRAY : BOOL
VAR_INPUT
	pData	:	POINTER TO WORD;
	Size	:	BYTE;
END_VAR
VAR
	i	:	BYTE := 0;
END_VAR
WHILE i<Size DO

	pData^ := 0;
	pData := pData + 1;
	i := i + 1;

END_WHILE
END_FUNCTION

(* POU ClevergyUtils/SHIFT_ARRAY, ST *)
FUNCTION SHIFT_ARRAY : BOOL
VAR_INPUT
	pData	:	POINTER TO ARRAY [1..2] OF WORD;
	Size	:	BYTE;
END_VAR
VAR
	pNew	:	POINTER TO WORD;
	i		:	BYTE;
END_VAR
(* Shift right *)
FOR i:=1 TO (Size-1) BY 1 DO

	(*pNew := pData + 1;*)
	pData^[i] := pData^[i+1];
	(*pData := pData + 1;*)

END_FOR
END_FUNCTION

(* POU GeoLumenWrapping/testFakeNodes, ST *)
FUNCTION testFakeNodes : BOOL
VAR_INPUT
END_VAR
VAR
	index:INT;
END_VAR
		FOR index:=5 TO MAX_LUXNUM DO
			TabListLux[index].xCoupled := TRUE; (*Indico che ho accoppiato l'ID con il mac address*)
			TabListLux[index].LuxID_Geolumen:=4; (*Salvo l'ID accoppiato al mac address - info che sarà poi da spedire al server*)
			LuxElement[index].ID := TabListLux[index].LuxNumber; (*  copio id del lux nella tabella delle variabili dei lux *)
			IF LuxElement[index].CTRL_MODE = 2 THEN
				(* init astro *)
				ASTR[index](ID:= LuxElement[index].ID, localTime:=Sys.Time_CT_DT);
				ASTR_CONFIG[index].ID:=ASTR[index].ID;
			END_IF
			LuxGeolumenNodes[index].ID_Geolumen:=TabListLux[index].LuxID_Geolumen;
			LuxGeolumenNodes[index].ID_Lux:=LuxElement[index].ID ;
		END_FOR
END_FUNCTION

(* POU ClevergyUtils/Word_Intero, ST *)
FUNCTION Word_Intero : INT
VAR_INPUT
	IN_WORD: WORD;
END_VAR
VAR
	Appoggio:DWORD;
END_VAR
IF IN_WORD>32766 THEN
	Appoggio:= (65534 - IN_WORD);
	Word_Intero:= -(DWORD_TO_INT(Appoggio));
ELSE
	Word_Intero:= WORD_TO_INT(IN_WORD);
END_IF
END_FUNCTION

(* Visualisation checkNodes
2 elements of other kinds (tables, trends, ...) not read
*)

(* Visualisation checkNodes_2
2 elements of other kinds (tables, trends, ...) not read
*)

(* Visualisation CMD_diagn
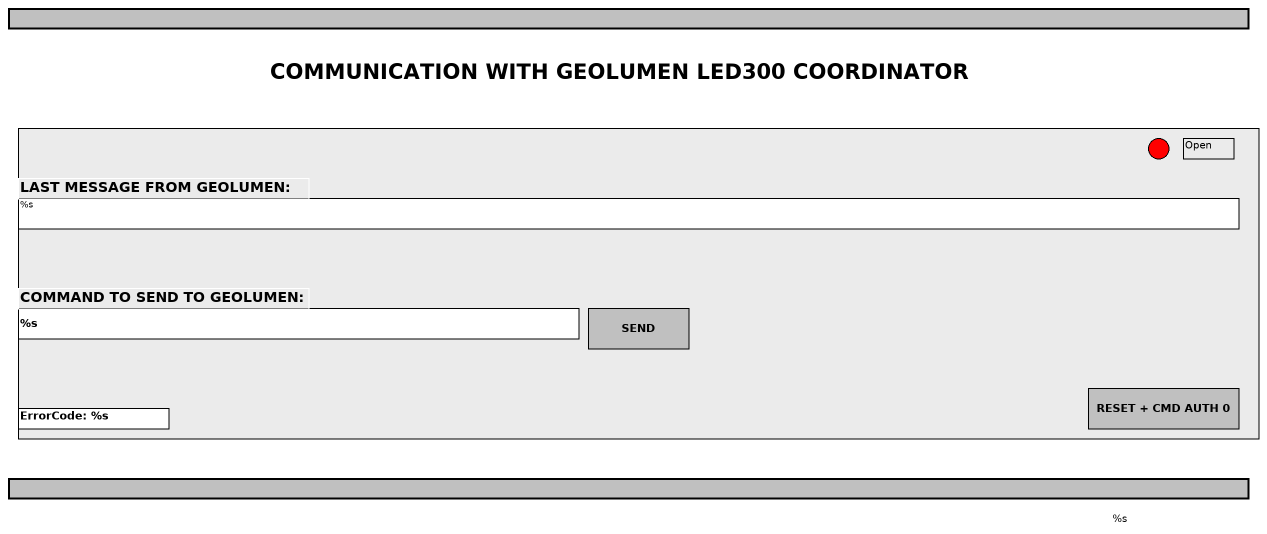
rectangle at (790,500)-(1131,521): text "%s"; shows Sys.Time_LogString
rectangle at (590,300)-(691,341): text "SEND"; runs INTERN ASSIGN LuxGeolumenDiagnostics.executeCommandRequest:=(TRUE)
rectangle at (270,50)-(971,81): text "COMMUNICATION WITH GEOLUMEN LED300 COORDINATOR"
rectangle at (20,300)-(581,331): text "%s"; shows LuxGeolumenDiagnostics.diagnosticCommand; editable
rectangle at (20,190)-(1241,221): text "%s"; shows obj_GeolumenCoordinator.LastMessage
rectangle at (20,400)-(171,421): text "ErrorCode: %s"; shows COM0.bError
rectangle at (1185,130)-(1236,151): text "Open"
ellipse at (1150,130)-(1171,151): alarm colour if COM0.COM_PORT_IST_OFFEN
rectangle at (20,170)-(311,191): text "LAST MESSAGE FROM GEOLUMEN:"
rectangle at (20,280)-(311,301): text "COMMAND TO SEND TO GEOLUMEN:"
rectangle at (1090,380)-(1241,421): text "RESET + CMD AUTH 0"; runs INTERN ASSIGN LuxGeolumenDiagnostics.executeCommandResetRequest:=(TRUE)
3 more shapes without text or variables
*)

